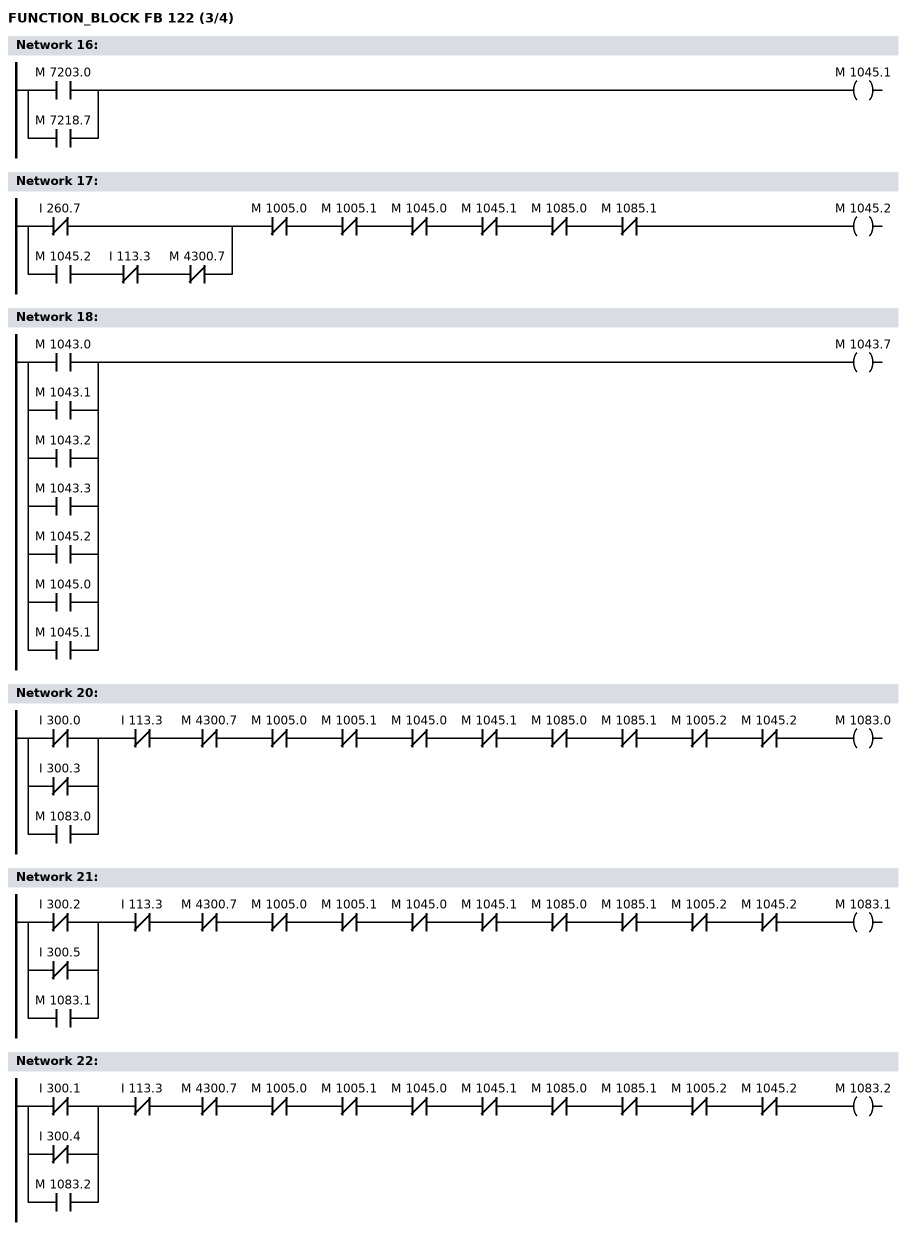

      O     M   7203.0;
      O     M   7218.7;
      =     M   1045.1;
NETWORK
TITLE =

      A(    ;
      ON    I    260.7;
      O     ;
      A     M   1045.2;
      AN    I    113.3;
      AN    M   4300.7;
      )     ;
      AN    M   1005.0;
      AN    M   1005.1;
      AN    M   1045.0;
      AN    M   1045.1;
      AN    M   1085.0;
      AN    M   1085.1;
      =     M   1045.2;
NETWORK
TITLE =

      O     M   1043.0;
      O     M   1043.1;
      O     M   1043.2;
      O     M   1043.3;
      O     M   1045.2;
      O     M   1045.0;
      O     M   1045.1;
      =     M   1043.7;
NETWORK
TITLE =리턴3 이상

NETWORK
TITLE =

      A(    ;
      ON    I    300.0;
      ON    I    300.3;
      O     M   1083.0;
      )     ;
      AN    I    113.3;
      AN    M   4300.7;
      AN    M   1005.0;
      AN    M   1005.1;
      AN    M   1045.0;
      AN    M   1045.1;
      AN    M   1085.0;
      AN    M   1085.1;
      AN    M   1005.2;
      AN    M   1045.2;
      =     M   1083.0;
NETWORK
TITLE =

      A(    ;
      ON    I    300.2;
      ON    I    300.5;
      O     M   1083.1;
      )     ;
      AN    I    113.3;
      AN    M   4300.7;
      AN    M   1005.0;
      AN    M   1005.1;
      AN    M   1045.0;
      AN    M   1045.1;
      AN    M   1085.0;
      AN    M   1085.1;
      AN    M   1005.2;
      AN    M   1045.2;
      =     M   1083.1;
NETWORK
TITLE =

      A(    ;
      ON    I    300.1;
      ON    I    300.4;
      O     M   1083.2;
      )     ;
      AN    I    113.3;
      AN    M   4300.7;
      AN    M   1005.0;
      AN    M   1005.1;
      AN    M   1045.0;
      AN    M   1045.1;
      AN    M   1085.0;
      AN    M   1085.1;
      AN    M   1005.2;
      AN    M   1045.2;
      =     M   1083.2;
NETWORK
TITLE =
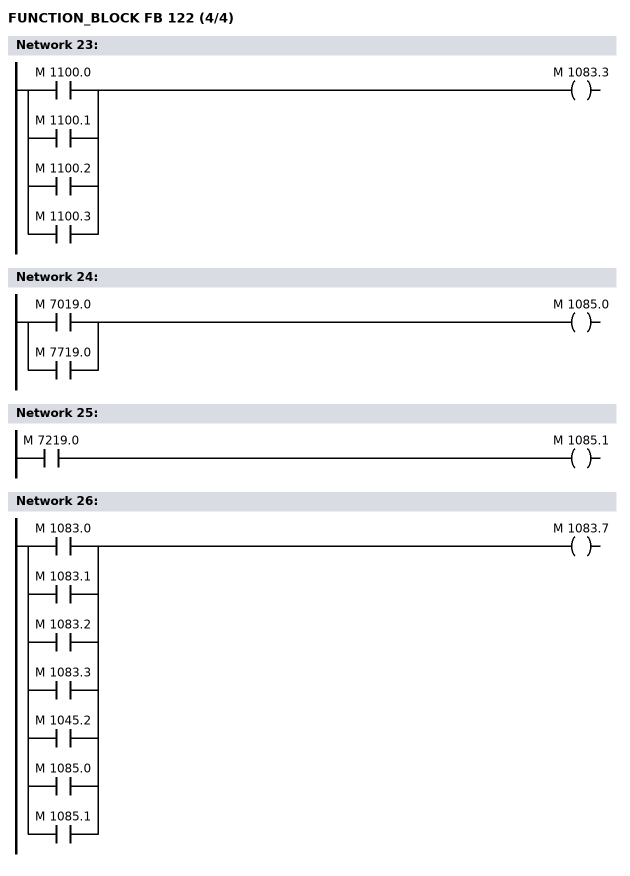

      O     M   1100.0;
      O     M   1100.1;
      O     M   1100.2;
      O     M   1100.3;
      =     M   1083.3;
NETWORK
TITLE =

      O     M   7019.0;
      O     M   7719.0;
      =     M   1085.0;
NETWORK
TITLE =

      A     M   7219.0;
      =     M   1085.1;
NETWORK
TITLE =

      O     M   1083.0;
      O     M   1083.1;
      O     M   1083.2;
      O     M   1083.3;
      O     M   1045.2;
      O     M   1085.0;
      O     M   1085.1;
      =     M   1083.7;
END_FUNCTION_BLOCK

DATA_BLOCK DB 122
TITLE =
VERSION : 0.0

 FB 122
BEGIN
END_DATA_BLOCK

FUNCTION FC 122 : VOID
TITLE =
VERSION : 0.1

BEGIN
NETWORK
TITLE =리턴1 SOL동작관련

NETWORK
TITLE =
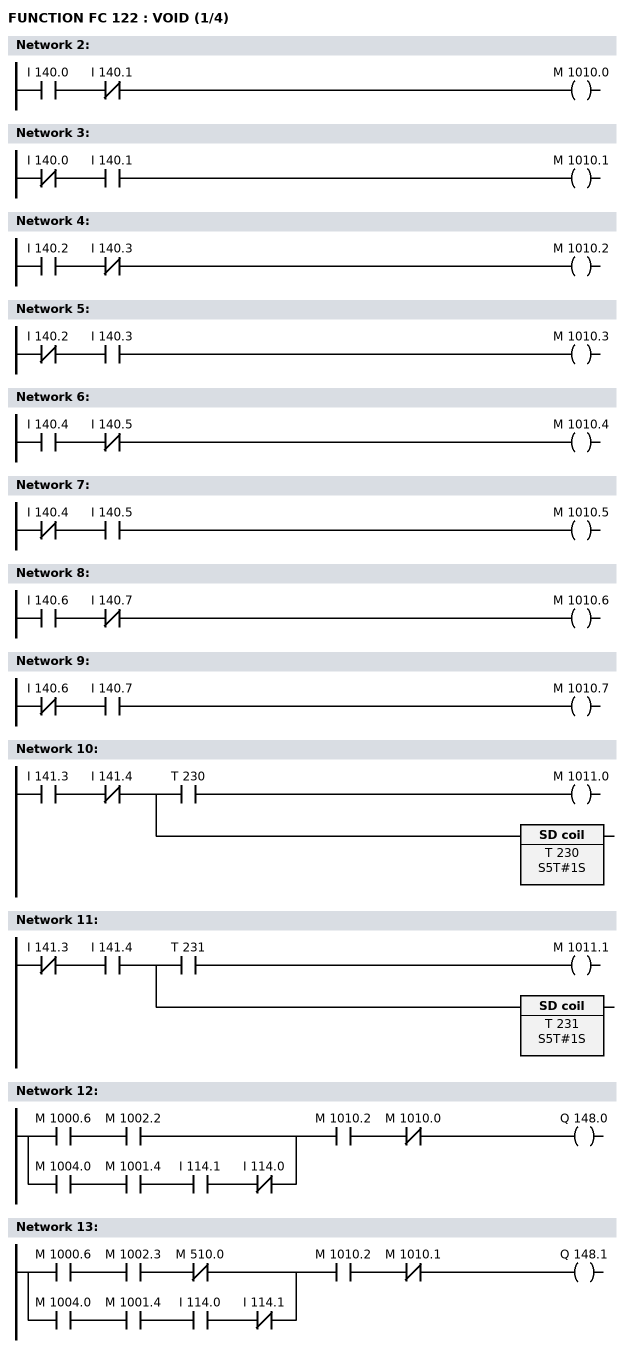

      A     I    140.0;
      AN    I    140.1;
      =     M   1010.0;
NETWORK
TITLE =

      AN    I    140.0;
      A     I    140.1;
      =     M   1010.1;
NETWORK
TITLE =

      A     I    140.2;
      AN    I    140.3;
      =     M   1010.2;
NETWORK
TITLE =

      AN    I    140.2;
      A     I    140.3;
      =     M   1010.3;
NETWORK
TITLE =

      A     I    140.4;
      AN    I    140.5;
      =     M   1010.4;
NETWORK
TITLE =

      AN    I    140.4;
      A     I    140.5;
      =     M   1010.5;
NETWORK
TITLE =

      A     I    140.6;
      AN    I    140.7;
      =     M   1010.6;
NETWORK
TITLE =

      AN    I    140.6;
      A     I    140.7;
      =     M   1010.7;
NETWORK
TITLE =

      A     I    141.3;
      AN    I    141.4;
      =     L      0.0;
      A     L      0.0;
      A     T    230;
      =     M   1011.0;
      A     L      0.0;
      BLD   102;
      L     S5T#1S;
      SD    T    230;
NETWORK
TITLE =

      AN    I    141.3;
      A     I    141.4;
      =     L      0.0;
      A     L      0.0;
      A     T    231;
      =     M   1011.1;
      A     L      0.0;
      BLD   102;
      L     S5T#1S;
      SD    T    231;
NETWORK
TITLE =

      A(    ;
      A     M   1000.6;
      A     M   1002.2;
      O     ;
      A     M   1004.0;
      A     M   1001.4;
      A     I    114.1;
      AN    I    114.0;
      )     ;
      A     M   1010.2;
      AN    M   1010.0;
      =     Q    148.0;
NETWORK
TITLE =

      A(    ;
      A     M   1000.6;
      A     M   1002.3;
      AN    M    510.0;
      O     ;
      A     M   1004.0;
      A     M   1001.4;
      A     I    114.0;
      AN    I    114.1;
      )     ;
      A     M   1010.2;
      AN    M   1010.1;
      =     Q    148.1;
NETWORK
TITLE =
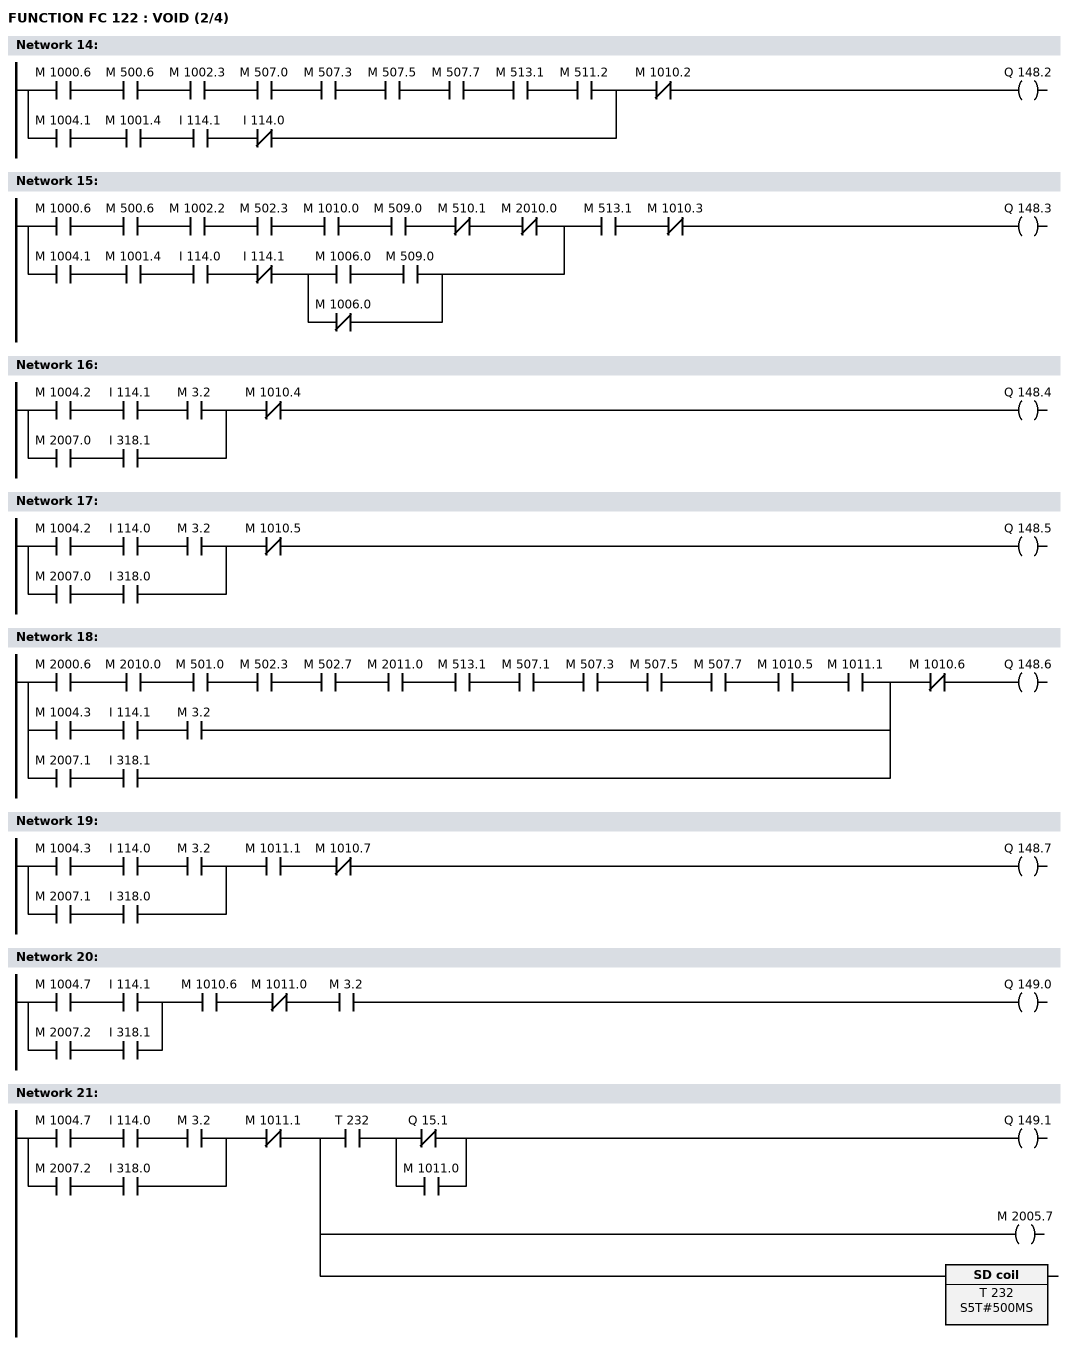

      A(    ;
      A     M   1000.6;
      A     M    500.6;
      A     M   1002.3;
      A     M    507.0;
      A     M    507.3;
      A     M    507.5;
      A     M    507.7;
      A     M    513.1;
      A     M    511.2;
      O     ;
      A     M   1004.1;
      A     M   1001.4;
      A     I    114.1;
      AN    I    114.0;
      )     ;
      AN    M   1010.2;
      =     Q    148.2;
NETWORK
TITLE =

      A(    ;
      A     M   1000.6;
      A     M    500.6;
      A     M   1002.2;
      A     M    502.3;
      A     M   1010.0;
      A     M    509.0;
      AN    M    510.1;
      AN    M   2010.0;
      O     ;
      A     M   1004.1;
      A     M   1001.4;
      A     I    114.0;
      AN    I    114.1;
      A(    ;
      A     M   1006.0;
      A     M    509.0;
      ON    M   1006.0;
      )     ;
      )     ;
      A     M    513.1;
      AN    M   1010.3;
      =     Q    148.3;
NETWORK
TITLE =

      A(    ;
      A     M   1004.2;
      A     I    114.1;
      A     M      3.2;
      O     ;
      A     M   2007.0;
      A     I    318.1;
      )     ;
      AN    M   1010.4;
      =     Q    148.4;
NETWORK
TITLE =

      A(    ;
      A     M   1004.2;
      A     I    114.0;
      A     M      3.2;
      O     ;
      A     M   2007.0;
      A     I    318.0;
      )     ;
      AN    M   1010.5;
      =     Q    148.5;
NETWORK
TITLE =

      A(    ;
      A     M   2000.6;
      A     M   2010.0;
      A     M    501.0;
      A     M    502.3;
      A     M    502.7;
      A     M   2011.0;
      A     M    513.1;
      A     M    507.1;
      A     M    507.3;
      A     M    507.5;
      A     M    507.7;
      A     M   1010.5;
      A     M   1011.1;
      O     ;
      A     M   1004.3;
      A     I    114.1;
      A     M      3.2;
      O     ;
      A     M   2007.1;
      A     I    318.1;
      )     ;
      AN    M   1010.6;
      =     Q    148.6;
NETWORK
TITLE =

      A(    ;
      A     M   1004.3;
      A     I    114.0;
      A     M      3.2;
      O     ;
      A     M   2007.1;
      A     I    318.0;
      )     ;
      A     M   1011.1;
      AN    M   1010.7;
      =     Q    148.7;
NETWORK
TITLE =

      A(    ;
      A     M   1004.7;
      A     I    114.1;
      O     ;
      A     M   2007.2;
      A     I    318.1;
      )     ;
      A     M   1010.6;
      AN    M   1011.0;
      A     M      3.2;
      =     Q    149.0;
NETWORK
TITLE =

      A(    ;
      A     M   1004.7;
      A     I    114.0;
      A     M      3.2;
      O     ;
      A     M   2007.2;
      A     I    318.0;
      )     ;
      AN    M   1011.1;
      =     L      0.0;
      A     L      0.0;
      A     T    232;
      A(    ;
      ON    Q     15.1;
      O     M   1011.0;
      )     ;
      =     Q    149.1;
      A     L      0.0;
      BLD   102;
      =     M   2005.7;
      A     L      0.0;
      BLD   102;
      L     S5T#500MS;
      SD    T    232;
NETWORK
TITLE =
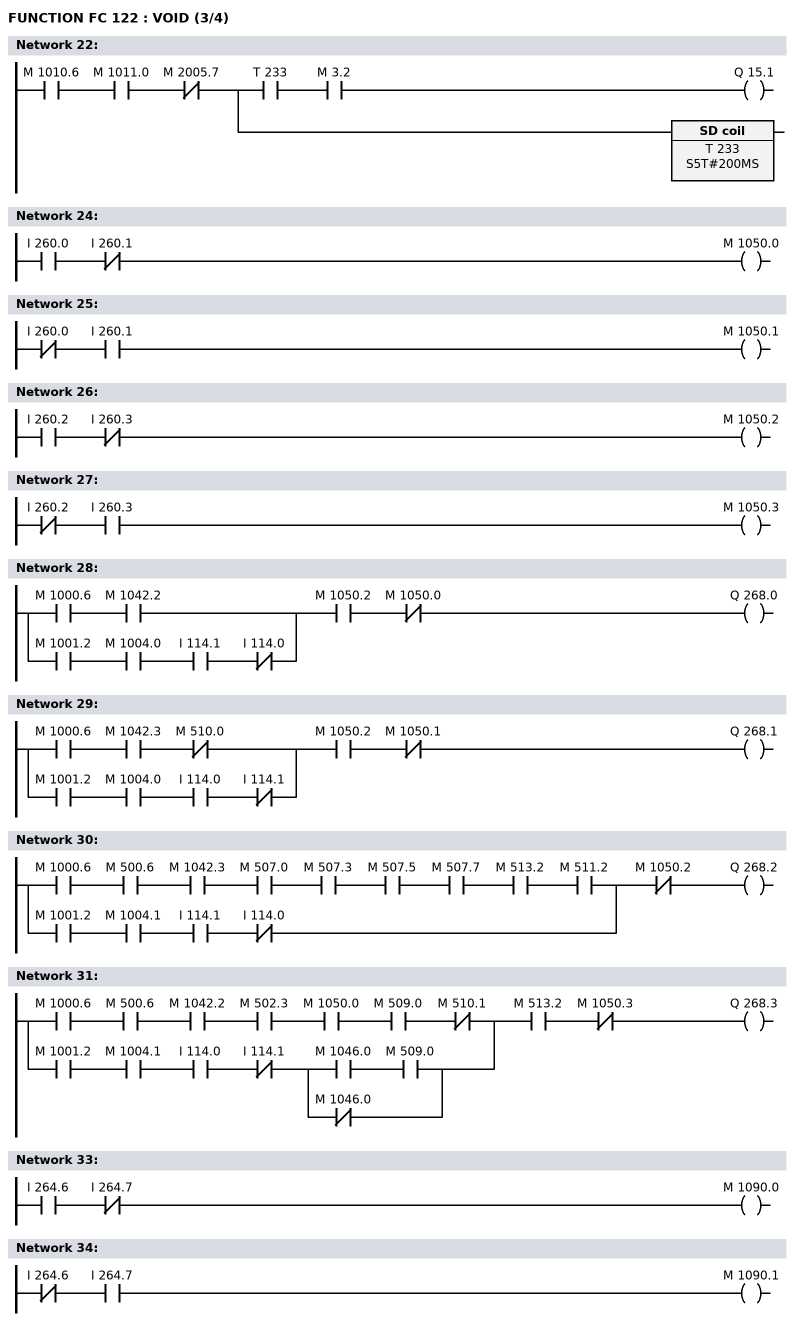

      A     M   1010.6;
      A     M   1011.0;
      AN    M   2005.7;
      =     L      0.0;
      A     L      0.0;
      A     T    233;
      A     M      3.2;
      =     Q     15.1;
      A     L      0.0;
      BLD   102;
      L     S5T#200MS;
      SD    T    233;
NETWORK
TITLE =RETURN2 SOL동작관련

NETWORK
TITLE =

      A     I    260.0;
      AN    I    260.1;
      =     M   1050.0;
NETWORK
TITLE =

      AN    I    260.0;
      A     I    260.1;
      =     M   1050.1;
NETWORK
TITLE =

      A     I    260.2;
      AN    I    260.3;
      =     M   1050.2;
NETWORK
TITLE =

      AN    I    260.2;
      A     I    260.3;
      =     M   1050.3;
NETWORK
TITLE =

      A(    ;
      A     M   1000.6;
      A     M   1042.2;
      O     ;
      A     M   1001.2;
      A     M   1004.0;
      A     I    114.1;
      AN    I    114.0;
      )     ;
      A     M   1050.2;
      AN    M   1050.0;
      =     Q    268.0;
NETWORK
TITLE =

      A(    ;
      A     M   1000.6;
      A     M   1042.3;
      AN    M    510.0;
      O     ;
      A     M   1001.2;
      A     M   1004.0;
      A     I    114.0;
      AN    I    114.1;
      )     ;
      A     M   1050.2;
      AN    M   1050.1;
      =     Q    268.1;
NETWORK
TITLE =

      A(    ;
      A     M   1000.6;
      A     M    500.6;
      A     M   1042.3;
      A     M    507.0;
      A     M    507.3;
      A     M    507.5;
      A     M    507.7;
      A     M    513.2;
      A     M    511.2;
      O     ;
      A     M   1001.2;
      A     M   1004.1;
      A     I    114.1;
      AN    I    114.0;
      )     ;
      AN    M   1050.2;
      =     Q    268.2;
NETWORK
TITLE =

      A(    ;
      A     M   1000.6;
      A     M    500.6;
      A     M   1042.2;
      A     M    502.3;
      A     M   1050.0;
      A     M    509.0;
      AN    M    510.1;
      O     ;
      A     M   1001.2;
      A     M   1004.1;
      A     I    114.0;
      AN    I    114.1;
      A(    ;
      A     M   1046.0;
      A     M    509.0;
      ON    M   1046.0;
      )     ;
      )     ;
      A     M    513.2;
      AN    M   1050.3;
      =     Q    268.3;
NETWORK
TITLE =RETURN3 SOL동작관련

NETWORK
TITLE =

      A     I    264.6;
      AN    I    264.7;
      =     M   1090.0;
NETWORK
TITLE =

      AN    I    264.6;
      A     I    264.7;
      =     M   1090.1;
NETWORK
TITLE =
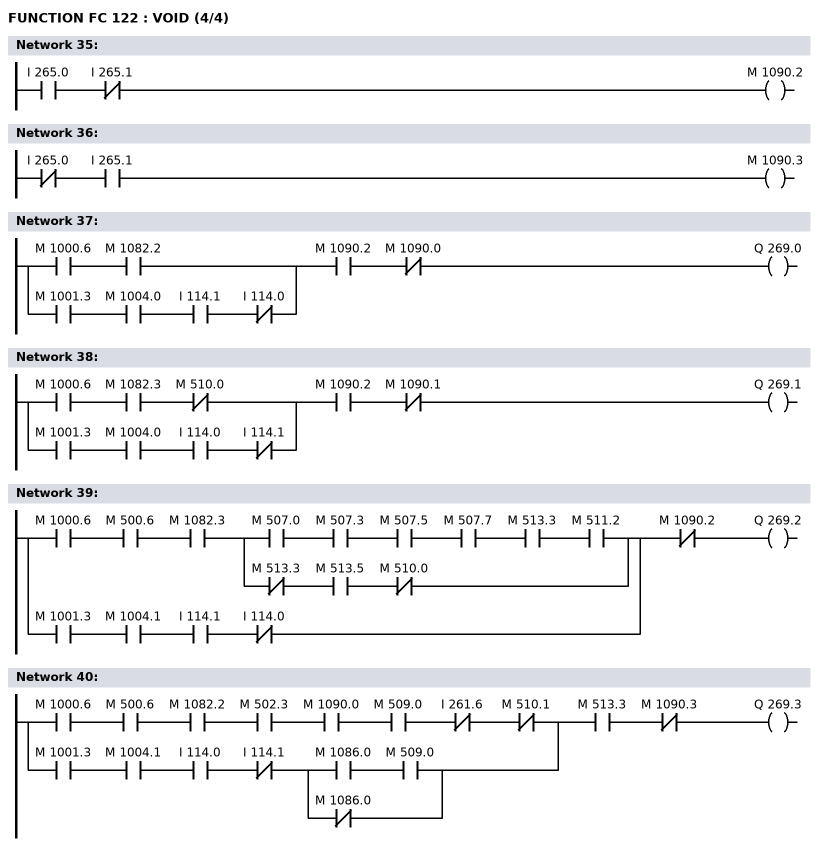

      A     I    265.0;
      AN    I    265.1;
      =     M   1090.2;
NETWORK
TITLE =

      AN    I    265.0;
      A     I    265.1;
      =     M   1090.3;
NETWORK
TITLE =

      A(    ;
      A     M   1000.6;
      A     M   1082.2;
      O     ;
      A     M   1001.3;
      A     M   1004.0;
      A     I    114.1;
      AN    I    114.0;
      )     ;
      A     M   1090.2;
      AN    M   1090.0;
      =     Q    269.0;
NETWORK
TITLE =

      A(    ;
      A     M   1000.6;
      A     M   1082.3;
      AN    M    510.0;
      O     ;
      A     M   1001.3;
      A     M   1004.0;
      A     I    114.0;
      AN    I    114.1;
      )     ;
      A     M   1090.2;
      AN    M   1090.1;
      =     Q    269.1;
NETWORK
TITLE =

      A(    ;
      A     M   1000.6;
      A     M    500.6;
      A     M   1082.3;
      A(    ;
      A     M    507.0;
      A     M    507.3;
      A     M    507.5;
      A     M    507.7;
      A     M    513.3;
      A     M    511.2;
      O     ;
      AN    M    513.3;
      A     M    513.5;
      AN    M    510.0;
      )     ;
      O     ;
      A     M   1001.3;
      A     M   1004.1;
      A     I    114.1;
      AN    I    114.0;
      )     ;
      AN    M   1090.2;
      =     Q    269.2;
NETWORK
TITLE =

      A(    ;
      A     M   1000.6;
      A     M    500.6;
      A     M   1082.2;
      A     M    502.3;
      A     M   1090.0;
      A     M    509.0;
      AN    I    261.6;
      AN    M    510.1;
      O     ;
      A     M   1001.3;
      A     M   1004.1;
      A     I    114.0;
      AN    I    114.1;
      A(    ;
      A     M   1086.0;
      A     M    509.0;
      ON    M   1086.0;
      )     ;
      )     ;
      A     M    513.3;
      AN    M   1090.3;
      =     Q    269.3;
END_FUNCTION

FUNCTION FC 123 : VOID
TITLE =
VERSION : 0.1

BEGIN
NETWORK
TITLE =
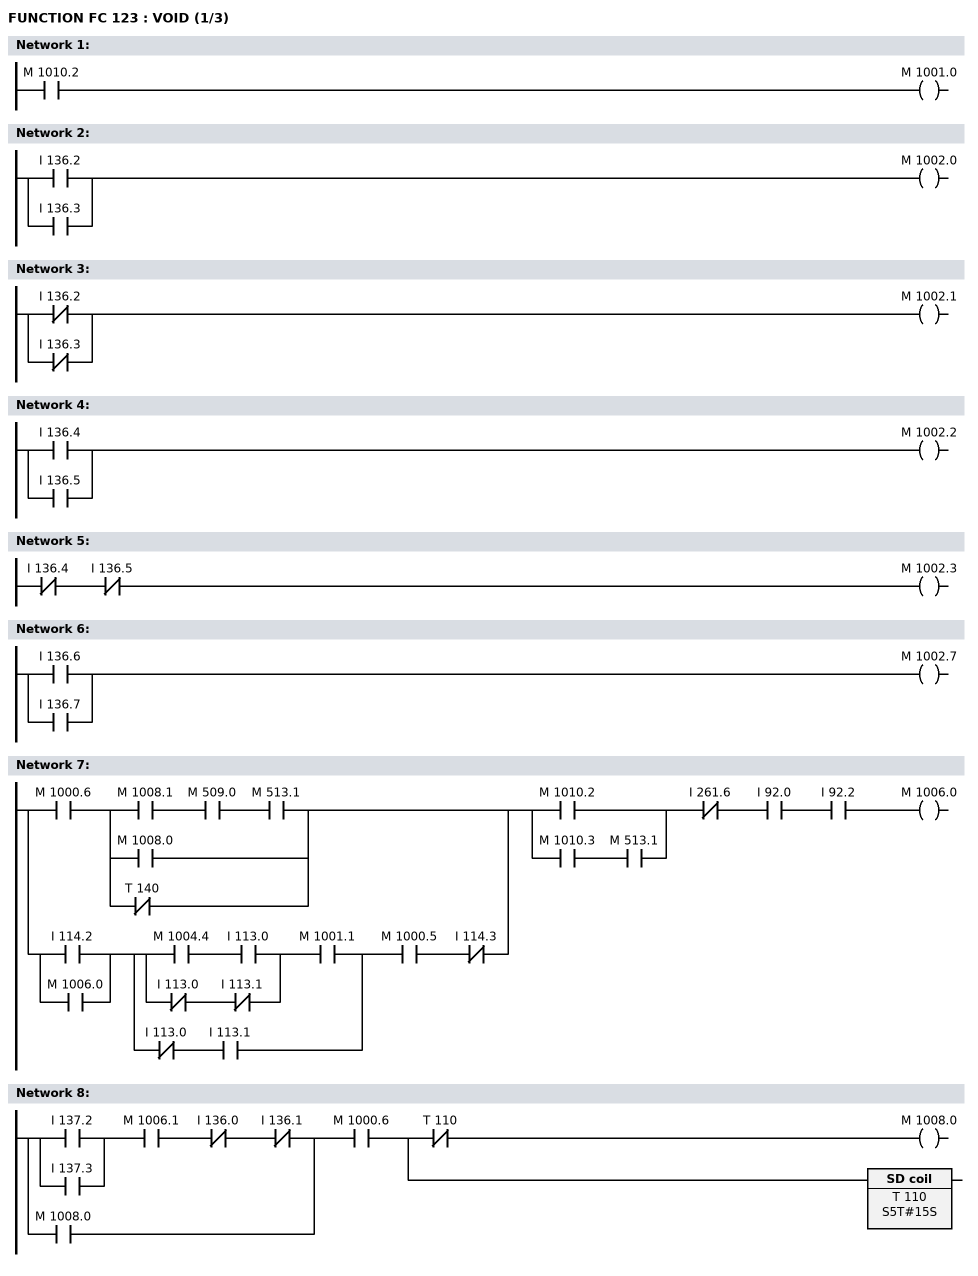

      A     M   1010.2;
      =     M   1001.0;
NETWORK
TITLE =

      O     I    136.2;
      O     I    136.3;
      =     M   1002.0;
NETWORK
TITLE =

      ON    I    136.2;
      ON    I    136.3;
      =     M   1002.1;
NETWORK
TITLE =

      O     I    136.4;
      O     I    136.5;
      =     M   1002.2;
NETWORK
TITLE =

      AN    I    136.4;
      AN    I    136.5;
      =     M   1002.3;
NETWORK
TITLE =

      O     I    136.6;
      O     I    136.7;
      =     M   1002.7;
NETWORK
TITLE =

      A(    ;
      A     M   1000.6;
      A(    ;
      A     M   1008.1;
      A     M    509.0;
      A     M    513.1;
      O     M   1008.0;
      ON    T    140;
      )     ;
      O     ;
      A(    ;
      O     I    114.2;
      O     M   1006.0;
      )     ;
      A(    ;
      A(    ;
      A     M   1004.4;
      A     I    113.0;
      O     ;
      AN    I    113.0;
      AN    I    113.1;
      )     ;
      A     M   1001.1;
      O     ;
      AN    I    113.0;
      A     I    113.1;
      )     ;
      A     M   1000.5;
      AN    I    114.3;
      )     ;
      A(    ;
      O     M   1010.2;
      O     ;
      A     M   1010.3;
      A     M    513.1;
      )     ;
      AN    I    261.6;
      A     I     92.0;
      A     I     92.2;
      =     M   1006.0;
NETWORK
TITLE =

      A(    ;
      A(    ;
      O     I    137.2;
      O     I    137.3;
      )     ;
      A     M   1006.1;
      AN    I    136.0;
      AN    I    136.1;
      O     M   1008.0;
      )     ;
      A     M   1000.6;
      =     L      0.0;
      A     L      0.0;
      AN    T    110;
      =     M   1008.0;
      A     L      0.0;
      BLD   102;
      L     S5T#15S;
      SD    T    110;
NETWORK
TITLE =
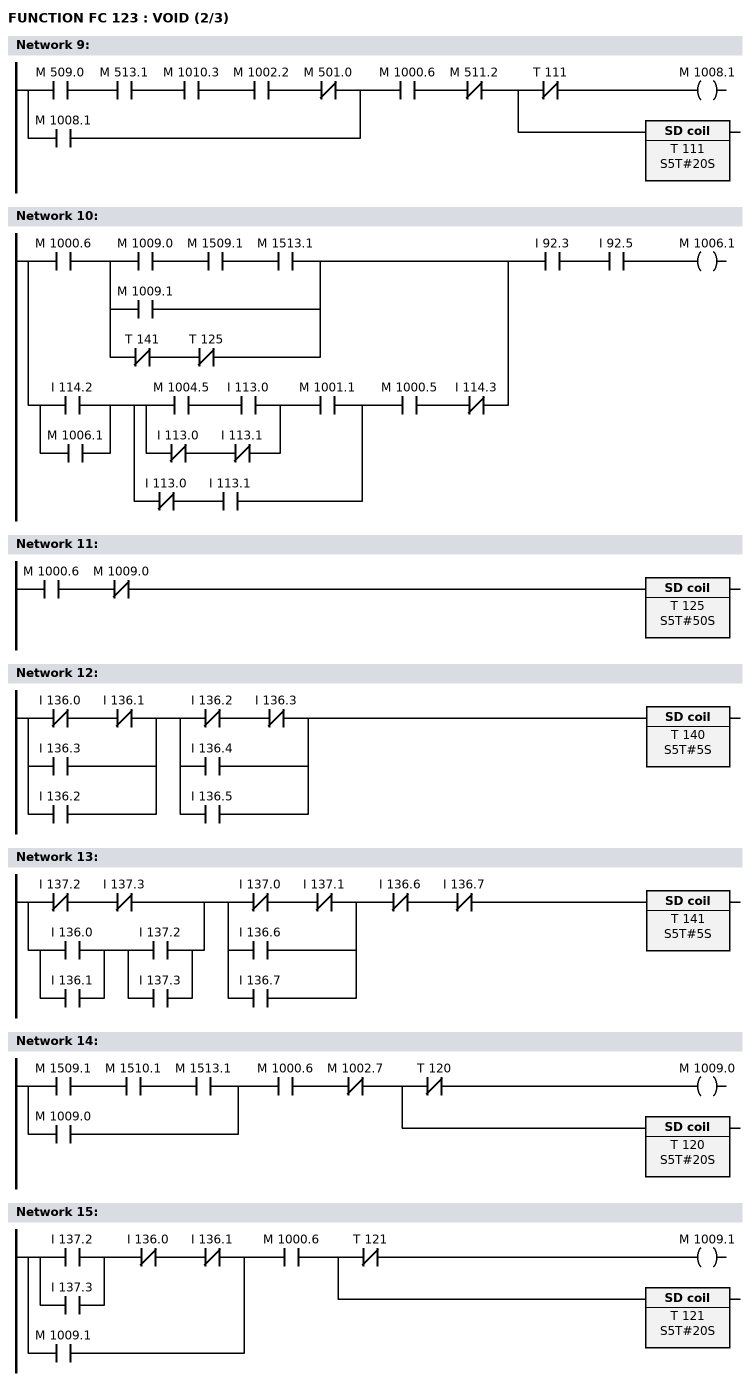

      A(    ;
      A     M    509.0;
      A     M    513.1;
      A     M   1010.3;
      A     M   1002.2;
      AN    M    501.0;
      O     M   1008.1;
      )     ;
      A     M   1000.6;
      AN    M    511.2;
      =     L      0.0;
      A     L      0.0;
      AN    T    111;
      =     M   1008.1;
      A     L      0.0;
      BLD   102;
      L     S5T#20S;
      SD    T    111;
NETWORK
TITLE =

      A(    ;
      A     M   1000.6;
      A(    ;
      A     M   1009.0;
      A     M   1509.1;
      A     M   1513.1;
      O     M   1009.1;
      O     ;
      AN    T    141;
      AN    T    125;
      )     ;
      O     ;
      A(    ;
      O     I    114.2;
      O     M   1006.1;
      )     ;
      A(    ;
      A(    ;
      A     M   1004.5;
      A     I    113.0;
      O     ;
      AN    I    113.0;
      AN    I    113.1;
      )     ;
      A     M   1001.1;
      O     ;
      AN    I    113.0;
      A     I    113.1;
      )     ;
      A     M   1000.5;
      AN    I    114.3;
      )     ;
      A     I     92.3;
      A     I     92.5;
      =     M   1006.1;
NETWORK
TITLE =

      A     M   1000.6;
      AN    M   1009.0;
      L     S5T#50S;
      SD    T    125;
NETWORK
TITLE =

      A(    ;
      AN    I    136.0;
      AN    I    136.1;
      O     I    136.3;
      O     I    136.2;
      )     ;
      A(    ;
      AN    I    136.2;
      AN    I    136.3;
      O     I    136.4;
      O     I    136.5;
      )     ;
      L     S5T#5S;
      SD    T    140;
NETWORK
TITLE =

      A(    ;
      AN    I    137.2;
      AN    I    137.3;
      O     ;
      A(    ;
      O     I    136.0;
      O     I    136.1;
      )     ;
      A(    ;
      O     I    137.2;
      O     I    137.3;
      )     ;
      )     ;
      A(    ;
      AN    I    137.0;
      AN    I    137.1;
      O     I    136.6;
      O     I    136.7;
      )     ;
      AN    I    136.6;
      AN    I    136.7;
      L     S5T#5S;
      SD    T    141;
NETWORK
TITLE =

      A(    ;
      A     M   1509.1;
      A     M   1510.1;
      A     M   1513.1;
      O     M   1009.0;
      )     ;
      A     M   1000.6;
      AN    M   1002.7;
      =     L      0.0;
      A     L      0.0;
      AN    T    120;
      =     M   1009.0;
      A     L      0.0;
      BLD   102;
      L     S5T#20S;
      SD    T    120;
NETWORK
TITLE =

      A(    ;
      A(    ;
      O     I    137.2;
      O     I    137.3;
      )     ;
      AN    I    136.0;
      AN    I    136.1;
      O     M   1009.1;
      )     ;
      A     M   1000.6;
      =     L      0.0;
      A     L      0.0;
      AN    T    121;
      =     M   1009.1;
      A     L      0.0;
      BLD   102;
      L     S5T#20S;
      SD    T    121;
NETWORK
TITLE =
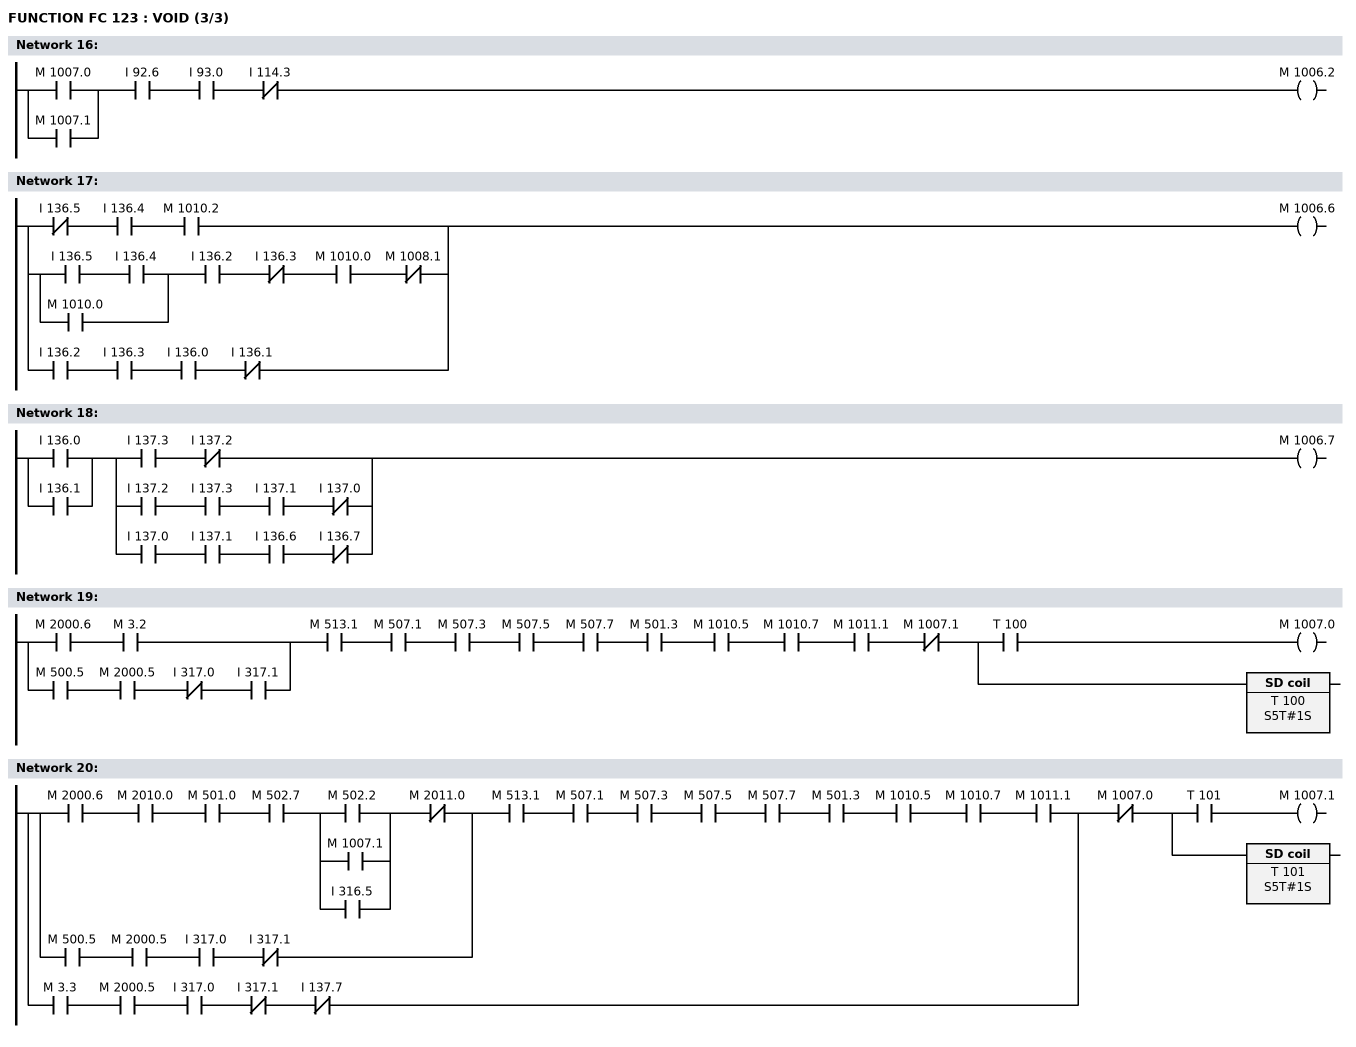

      A(    ;
      O     M   1007.0;
      O     M   1007.1;
      )     ;
      A     I     92.6;
      A     I     93.0;
      AN    I    114.3;
      =     M   1006.2;
NETWORK
TITLE =

      AN    I    136.5;
      A     I    136.4;
      A     M   1010.2;
      O     ;
      A(    ;
      A     I    136.5;
      A     I    136.4;
      O     M   1010.0;
      )     ;
      A     I    136.2;
      AN    I    136.3;
      A     M   1010.0;
      AN    M   1008.1;
      O     ;
      A     I    136.2;
      A     I    136.3;
      A     I    136.0;
      AN    I    136.1;
      =     M   1006.6;
NETWORK
TITLE =

      A(    ;
      O     I    136.0;
      O     I    136.1;
      )     ;
      A(    ;
      A     I    137.3;
      AN    I    137.2;
      O     ;
      A     I    137.2;
      A     I    137.3;
      A     I    137.1;
      AN    I    137.0;
      O     ;
      A     I    137.0;
      A     I    137.1;
      A     I    136.6;
      AN    I    136.7;
      )     ;
      =     M   1006.7;
NETWORK
TITLE =

      A(    ;
      A     M   2000.6;
      A     M      3.2;
      O     ;
      A     M    500.5;
      A     M   2000.5;
      AN    I    317.0;
      A     I    317.1;
      )     ;
      A     M    513.1;
      A     M    507.1;
      A     M    507.3;
      A     M    507.5;
      A     M    507.7;
      A     M    501.3;
      A     M   1010.5;
      A     M   1010.7;
      A     M   1011.1;
      AN    M   1007.1;
      =     L      0.0;
      A     L      0.0;
      A     T    100;
      =     M   1007.0;
      A     L      0.0;
      BLD   102;
      L     S5T#1S;
      SD    T    100;
NETWORK
TITLE =

      A(    ;
      A(    ;
      A     M   2000.6;
      A     M   2010.0;
      A     M    501.0;
      A     M    502.7;
      A(    ;
      O     M    502.2;
      O     M   1007.1;
      O     I    316.5;
      )     ;
      AN    M   2011.0;
      O     ;
      A     M    500.5;
      A     M   2000.5;
      A     I    317.0;
      AN    I    317.1;
      )     ;
      A     M    513.1;
      A     M    507.1;
      A     M    507.3;
      A     M    507.5;
      A     M    507.7;
      A     M    501.3;
      A     M   1010.5;
      A     M   1010.7;
      A     M   1011.1;
      O     ;
      A     M      3.3;
      A     M   2000.5;
      A     I    317.0;
      AN    I    317.1;
      AN    I    137.7;
      )     ;
      AN    M   1007.0;
      =     L      0.0;
      A     L      0.0;
      A     T    101;
      =     M   1007.1;
      A     L      0.0;
      BLD   102;
      L     S5T#1S;
      SD    T    101;
END_FUNCTION

FUNCTION FC 124 : VOID
TITLE =
VERSION : 0.1

BEGIN
NETWORK
TITLE =
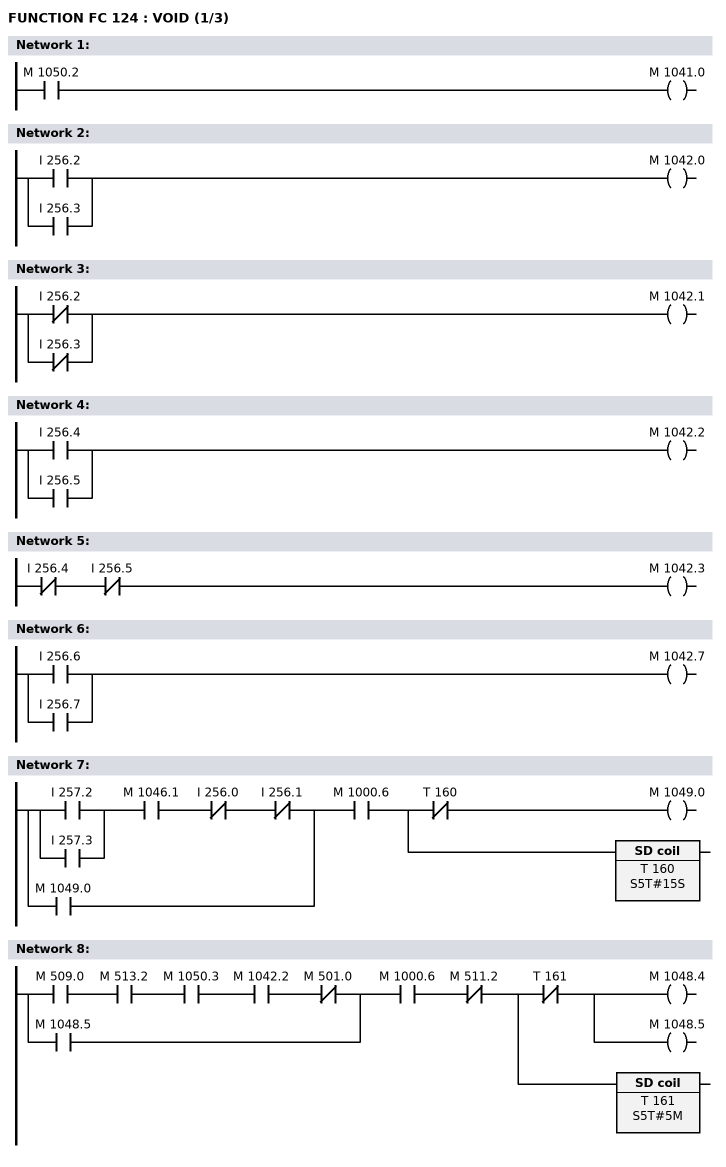

      A     M   1050.2;
      =     M   1041.0;
NETWORK
TITLE =

      O     I    256.2;
      O     I    256.3;
      =     M   1042.0;
NETWORK
TITLE =

      ON    I    256.2;
      ON    I    256.3;
      =     M   1042.1;
NETWORK
TITLE =

      O     I    256.4;
      O     I    256.5;
      =     M   1042.2;
NETWORK
TITLE =

      AN    I    256.4;
      AN    I    256.5;
      =     M   1042.3;
NETWORK
TITLE =

      O     I    256.6;
      O     I    256.7;
      =     M   1042.7;
NETWORK
TITLE =

      A(    ;
      A(    ;
      O     I    257.2;
      O     I    257.3;
      )     ;
      A     M   1046.1;
      AN    I    256.0;
      AN    I    256.1;
      O     M   1049.0;
      )     ;
      A     M   1000.6;
      =     L      0.0;
      A     L      0.0;
      AN    T    160;
      =     M   1049.0;
      A     L      0.0;
      BLD   102;
      L     S5T#15S;
      SD    T    160;
NETWORK
TITLE =

      A(    ;
      A     M    509.0;
      A     M    513.2;
      A     M   1050.3;
      A     M   1042.2;
      AN    M    501.0;
      O     M   1048.5;
      )     ;
      A     M   1000.6;
      AN    M    511.2;
      =     L      0.0;
      A     L      0.0;
      AN    T    161;
      =     M   1048.4;
      =     M   1048.5;
      A     L      0.0;
      BLD   102;
      L     S5T#5M;
      SD    T    161;
NETWORK
TITLE =
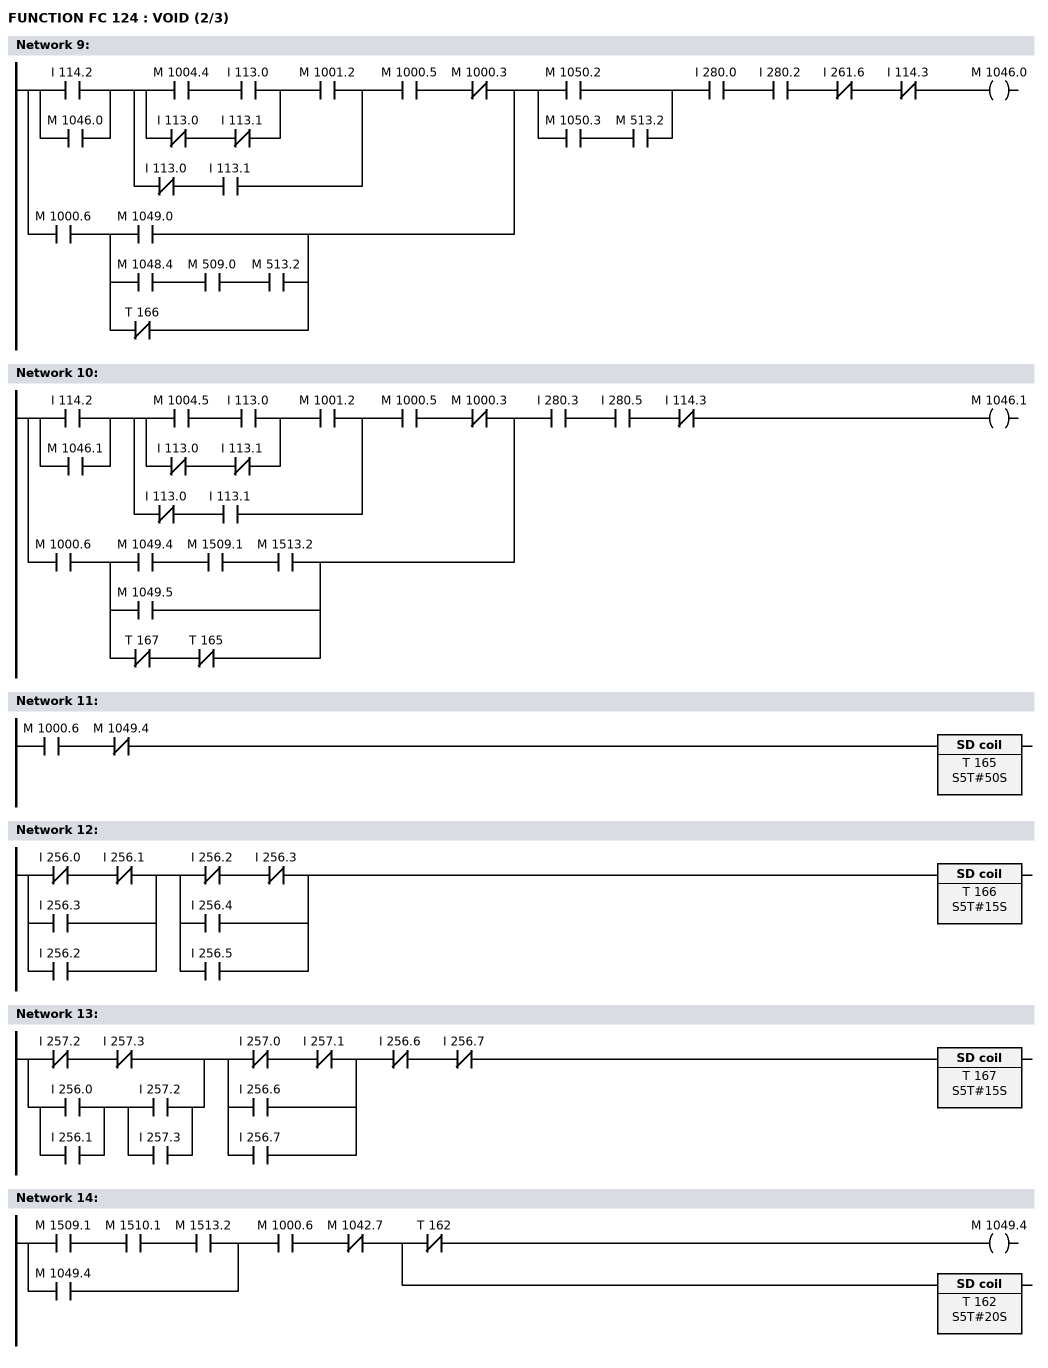

      A(    ;
      A(    ;
      O     I    114.2;
      O     M   1046.0;
      )     ;
      A(    ;
      A(    ;
      A     M   1004.4;
      A     I    113.0;
      O     ;
      AN    I    113.0;
      AN    I    113.1;
      )     ;
      A     M   1001.2;
      O     ;
      AN    I    113.0;
      A     I    113.1;
      )     ;
      A     M   1000.5;
      AN    M   1000.3;
      O     ;
      A     M   1000.6;
      A(    ;
      O     M   1049.0;
      O     ;
      A     M   1048.4;
      A     M    509.0;
      A     M    513.2;
      ON    T    166;
      )     ;
      )     ;
      A(    ;
      O     M   1050.2;
      O     ;
      A     M   1050.3;
      A     M    513.2;
      )     ;
      A     I    280.0;
      A     I    280.2;
      AN    I    261.6;
      AN    I    114.3;
      =     M   1046.0;
NETWORK
TITLE =

      A(    ;
      A(    ;
      O     I    114.2;
      O     M   1046.1;
      )     ;
      A(    ;
      A(    ;
      A     M   1004.5;
      A     I    113.0;
      O     ;
      AN    I    113.0;
      AN    I    113.1;
      )     ;
      A     M   1001.2;
      O     ;
      AN    I    113.0;
      A     I    113.1;
      )     ;
      A     M   1000.5;
      AN    M   1000.3;
      O     ;
      A     M   1000.6;
      A(    ;
      A     M   1049.4;
      A     M   1509.1;
      A     M   1513.2;
      O     M   1049.5;
      O     ;
      AN    T    167;
      AN    T    165;
      )     ;
      )     ;
      A     I    280.3;
      A     I    280.5;
      AN    I    114.3;
      =     M   1046.1;
NETWORK
TITLE =

      A     M   1000.6;
      AN    M   1049.4;
      L     S5T#50S;
      SD    T    165;
NETWORK
TITLE =

      A(    ;
      AN    I    256.0;
      AN    I    256.1;
      O     I    256.3;
      O     I    256.2;
      )     ;
      A(    ;
      AN    I    256.2;
      AN    I    256.3;
      O     I    256.4;
      O     I    256.5;
      )     ;
      L     S5T#15S;
      SD    T    166;
NETWORK
TITLE =

      A(    ;
      AN    I    257.2;
      AN    I    257.3;
      O     ;
      A(    ;
      O     I    256.0;
      O     I    256.1;
      )     ;
      A(    ;
      O     I    257.2;
      O     I    257.3;
      )     ;
      )     ;
      A(    ;
      AN    I    257.0;
      AN    I    257.1;
      O     I    256.6;
      O     I    256.7;
      )     ;
      AN    I    256.6;
      AN    I    256.7;
      L     S5T#15S;
      SD    T    167;
NETWORK
TITLE =

      A(    ;
      A     M   1509.1;
      A     M   1510.1;
      A     M   1513.2;
      O     M   1049.4;
      )     ;
      A     M   1000.6;
      AN    M   1042.7;
      =     L      0.0;
      A     L      0.0;
      AN    T    162;
      =     M   1049.4;
      A     L      0.0;
      BLD   102;
      L     S5T#20S;
      SD    T    162;
NETWORK
TITLE =
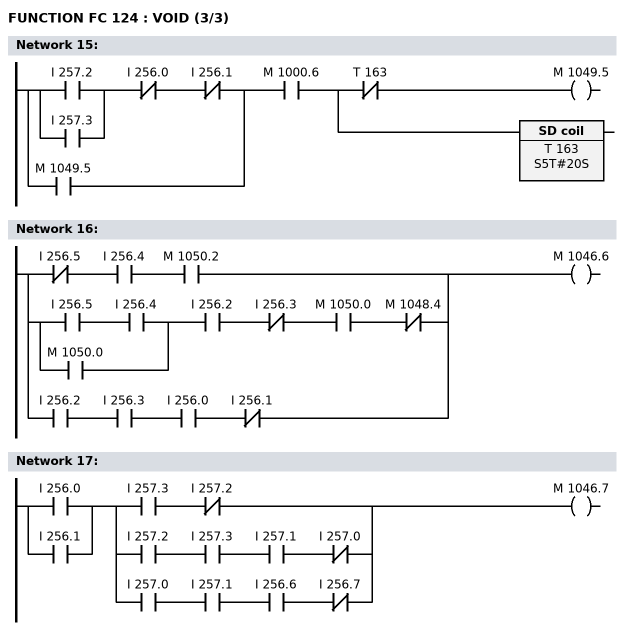

      A(    ;
      A(    ;
      O     I    257.2;
      O     I    257.3;
      )     ;
      AN    I    256.0;
      AN    I    256.1;
      O     M   1049.5;
      )     ;
      A     M   1000.6;
      =     L      0.0;
      A     L      0.0;
      AN    T    163;
      =     M   1049.5;
      A     L      0.0;
      BLD   102;
      L     S5T#20S;
      SD    T    163;
NETWORK
TITLE =

      AN    I    256.5;
      A     I    256.4;
      A     M   1050.2;
      O     ;
      A(    ;
      A     I    256.5;
      A     I    256.4;
      O     M   1050.0;
      )     ;
      A     I    256.2;
      AN    I    256.3;
      A     M   1050.0;
      AN    M   1048.4;
      O     ;
      A     I    256.2;
      A     I    256.3;
      A     I    256.0;
      AN    I    256.1;
      =     M   1046.6;
NETWORK
TITLE =

      A(    ;
      O     I    256.0;
      O     I    256.1;
      )     ;
      A(    ;
      A     I    257.3;
      AN    I    257.2;
      O     ;
      A     I    257.2;
      A     I    257.3;
      A     I    257.1;
      AN    I    257.0;
      O     ;
      A     I    257.0;
      A     I    257.1;
      A     I    256.6;
      AN    I    256.7;
      )     ;
      =     M   1046.7;
END_FUNCTION

FUNCTION FC 125 : VOID
TITLE =
VERSION : 0.1

BEGIN
NETWORK
TITLE =
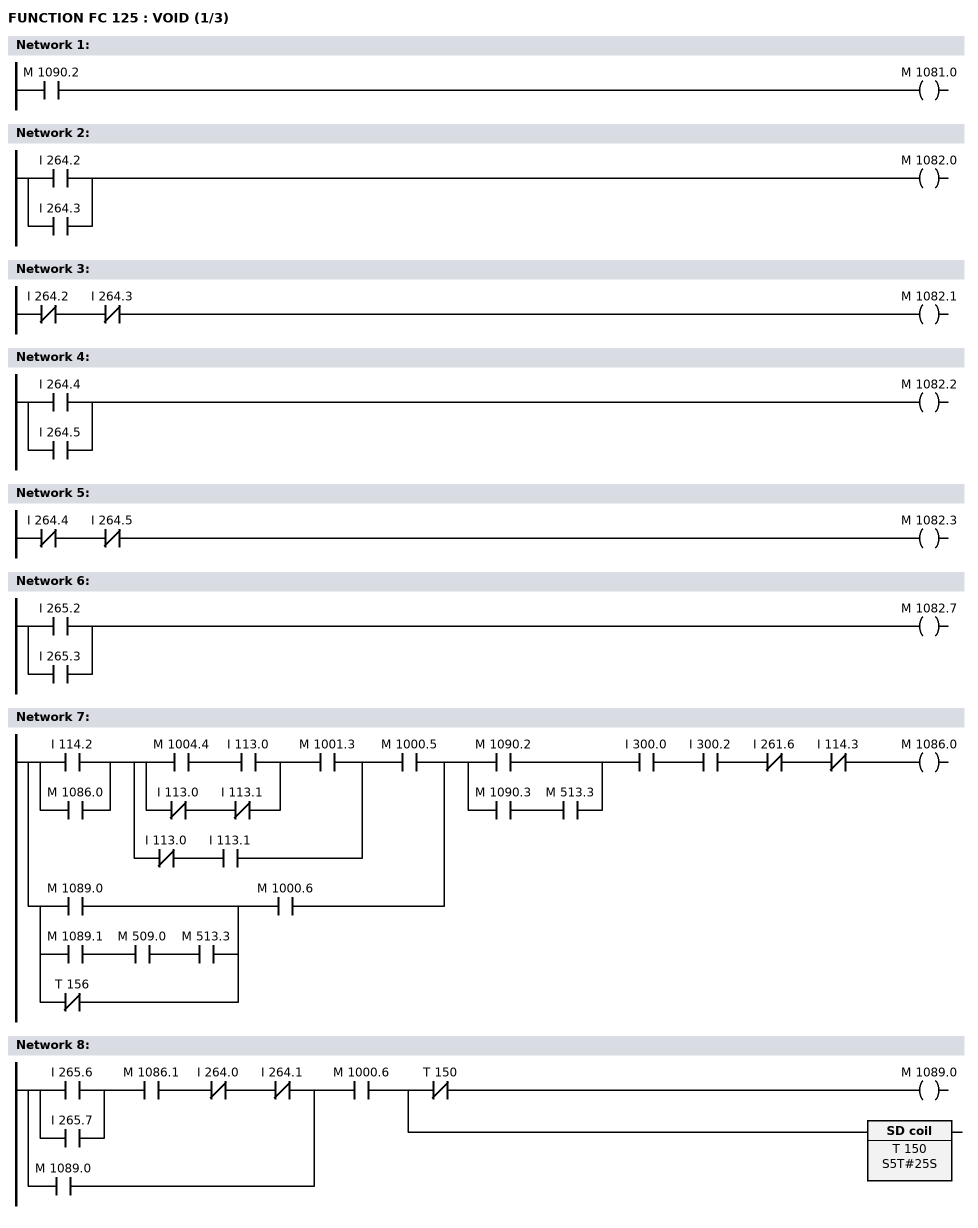

      A     M   1090.2;
      =     M   1081.0;
NETWORK
TITLE =

      O     I    264.2;
      O     I    264.3;
      =     M   1082.0;
NETWORK
TITLE =

      AN    I    264.2;
      AN    I    264.3;
      =     M   1082.1;
NETWORK
TITLE =

      O     I    264.4;
      O     I    264.5;
      =     M   1082.2;
NETWORK
TITLE =

      AN    I    264.4;
      AN    I    264.5;
      =     M   1082.3;
NETWORK
TITLE =

      O     I    265.2;
      O     I    265.3;
      =     M   1082.7;
NETWORK
TITLE =

      A(    ;
      A(    ;
      O     I    114.2;
      O     M   1086.0;
      )     ;
      A(    ;
      A(    ;
      A     M   1004.4;
      A     I    113.0;
      O     ;
      AN    I    113.0;
      AN    I    113.1;
      )     ;
      A     M   1001.3;
      O     ;
      AN    I    113.0;
      A     I    113.1;
      )     ;
      A     M   1000.5;
      O     ;
      A(    ;
      O     M   1089.0;
      O     ;
      A     M   1089.1;
      A     M    509.0;
      A     M    513.3;
      ON    T    156;
      )     ;
      A     M   1000.6;
      )     ;
      A(    ;
      O     M   1090.2;
      O     ;
      A     M   1090.3;
      A     M    513.3;
      )     ;
      A     I    300.0;
      A     I    300.2;
      AN    I    261.6;
      AN    I    114.3;
      =     M   1086.0;
NETWORK
TITLE =

      A(    ;
      A(    ;
      O     I    265.6;
      O     I    265.7;
      )     ;
      A     M   1086.1;
      AN    I    264.0;
      AN    I    264.1;
      O     M   1089.0;
      )     ;
      A     M   1000.6;
      =     L      0.0;
      A     L      0.0;
      AN    T    150;
      =     M   1089.0;
      A     L      0.0;
      BLD   102;
      L     S5T#25S;
      SD    T    150;
NETWORK
TITLE =
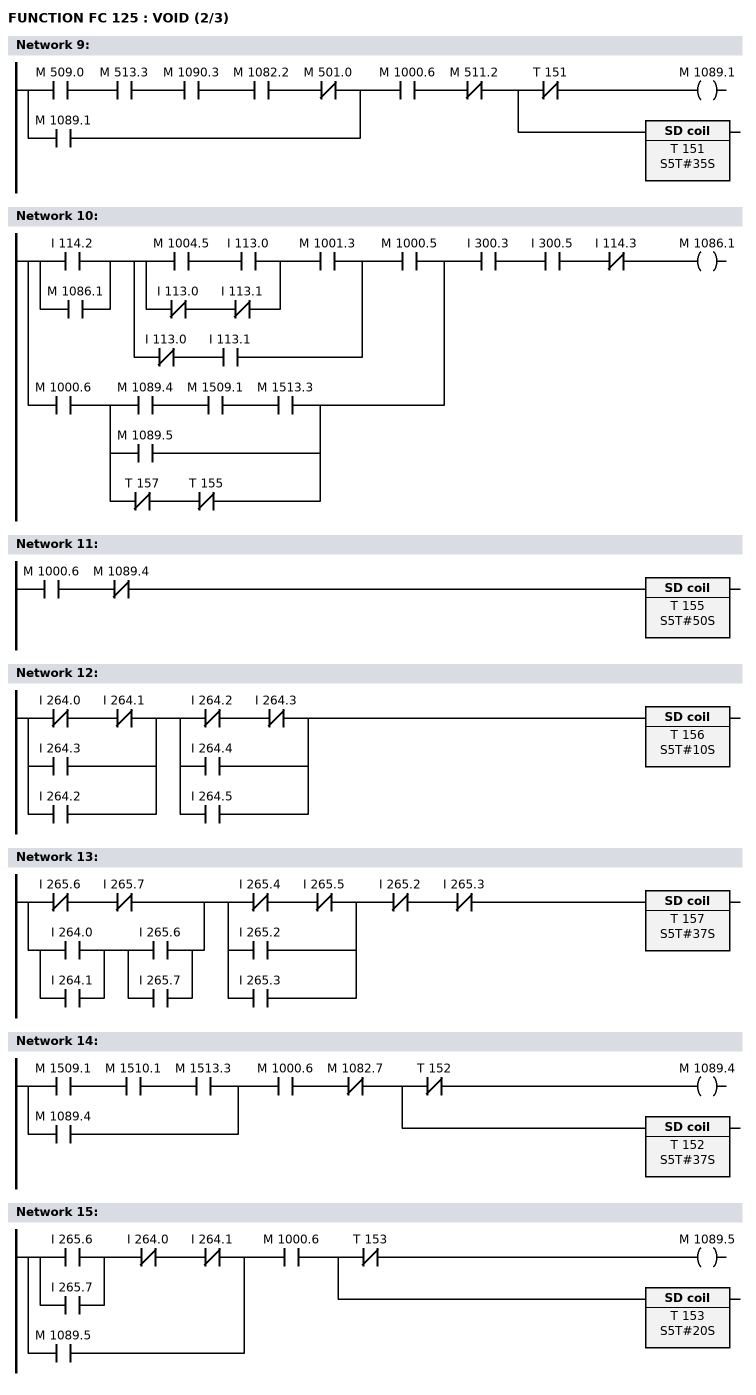

      A(    ;
      A     M    509.0;
      A     M    513.3;
      A     M   1090.3;
      A     M   1082.2;
      AN    M    501.0;
      O     M   1089.1;
      )     ;
      A     M   1000.6;
      AN    M    511.2;
      =     L      0.0;
      A     L      0.0;
      AN    T    151;
      =     M   1089.1;
      A     L      0.0;
      BLD   102;
      L     S5T#35S;
      SD    T    151;
NETWORK
TITLE =

      A(    ;
      A(    ;
      O     I    114.2;
      O     M   1086.1;
      )     ;
      A(    ;
      A(    ;
      A     M   1004.5;
      A     I    113.0;
      O     ;
      AN    I    113.0;
      AN    I    113.1;
      )     ;
      A     M   1001.3;
      O     ;
      AN    I    113.0;
      A     I    113.1;
      )     ;
      A     M   1000.5;
      O     ;
      A     M   1000.6;
      A(    ;
      A     M   1089.4;
      A     M   1509.1;
      A     M   1513.3;
      O     M   1089.5;
      O     ;
      AN    T    157;
      AN    T    155;
      )     ;
      )     ;
      A     I    300.3;
      A     I    300.5;
      AN    I    114.3;
      =     M   1086.1;
NETWORK
TITLE =

      A     M   1000.6;
      AN    M   1089.4;
      L     S5T#50S;
      SD    T    155;
NETWORK
TITLE =

      A(    ;
      AN    I    264.0;
      AN    I    264.1;
      O     I    264.3;
      O     I    264.2;
      )     ;
      A(    ;
      AN    I    264.2;
      AN    I    264.3;
      O     I    264.4;
      O     I    264.5;
      )     ;
      L     S5T#10S;
      SD    T    156;
NETWORK
TITLE =

      A(    ;
      AN    I    265.6;
      AN    I    265.7;
      O     ;
      A(    ;
      O     I    264.0;
      O     I    264.1;
      )     ;
      A(    ;
      O     I    265.6;
      O     I    265.7;
      )     ;
      )     ;
      A(    ;
      AN    I    265.4;
      AN    I    265.5;
      O     I    265.2;
      O     I    265.3;
      )     ;
      AN    I    265.2;
      AN    I    265.3;
      L     S5T#37S;
      SD    T    157;
NETWORK
TITLE =

      A(    ;
      A     M   1509.1;
      A     M   1510.1;
      A     M   1513.3;
      O     M   1089.4;
      )     ;
      A     M   1000.6;
      AN    M   1082.7;
      =     L      0.0;
      A     L      0.0;
      AN    T    152;
      =     M   1089.4;
      A     L      0.0;
      BLD   102;
      L     S5T#37S;
      SD    T    152;
NETWORK
TITLE =

      A(    ;
      A(    ;
      O     I    265.6;
      O     I    265.7;
      )     ;
      AN    I    264.0;
      AN    I    264.1;
      O     M   1089.5;
      )     ;
      A     M   1000.6;
      =     L      0.0;
      A     L      0.0;
      AN    T    153;
      =     M   1089.5;
      A     L      0.0;
      BLD   102;
      L     S5T#20S;
      SD    T    153;
NETWORK
TITLE =
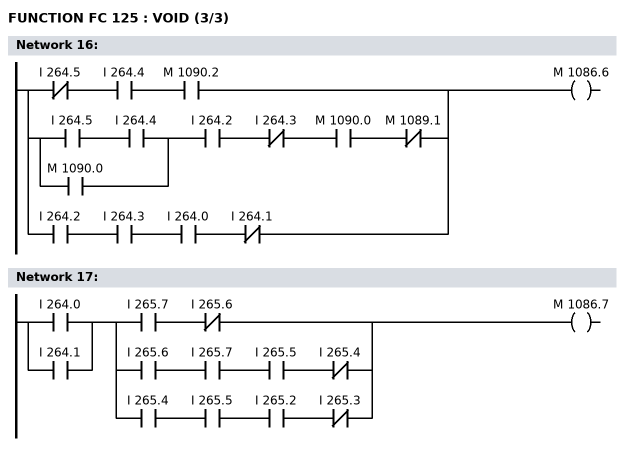

      AN    I    264.5;
      A     I    264.4;
      A     M   1090.2;
      O     ;
      A(    ;
      A     I    264.5;
      A     I    264.4;
      O     M   1090.0;
      )     ;
      A     I    264.2;
      AN    I    264.3;
      A     M   1090.0;
      AN    M   1089.1;
      O     ;
      A     I    264.2;
      A     I    264.3;
      A     I    264.0;
      AN    I    264.1;
      =     M   1086.6;
NETWORK
TITLE =

      A(    ;
      O     I    264.0;
      O     I    264.1;
      )     ;
      A(    ;
      A     I    265.7;
      AN    I    265.6;
      O     ;
      A     I    265.6;
      A     I    265.7;
      A     I    265.5;
      AN    I    265.4;
      O     ;
      A     I    265.4;
      A     I    265.5;
      A     I    265.2;
      AN    I    265.3;
      )     ;
      =     M   1086.7;
END_FUNCTION

FUNCTION FC 126 : VOID
TITLE =
VERSION : 0.1

BEGIN
NETWORK
TITLE =리턴1 인버터 인터록

NETWORK
TITLE =
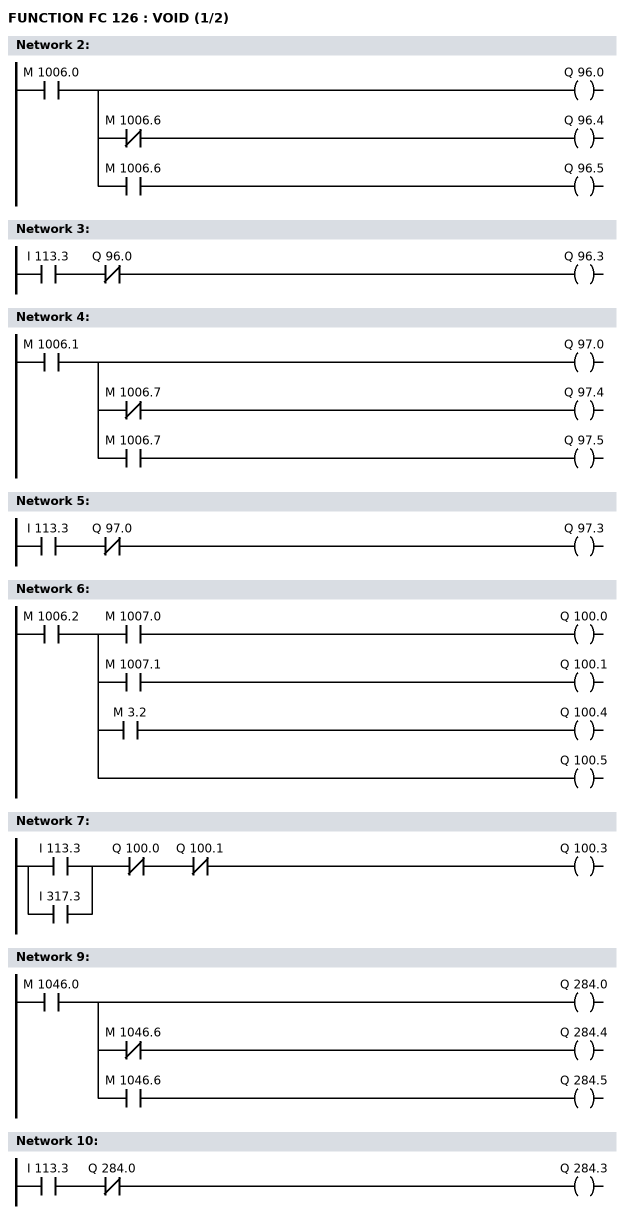

      A     M   1006.0;
      =     L      0.0;
      A     L      0.0;
      BLD   102;
      =     Q     96.0;
      A     L      0.0;
      AN    M   1006.6;
      =     Q     96.4;
      A     L      0.0;
      A     M   1006.6;
      =     Q     96.5;
NETWORK
TITLE =

      A     I    113.3;
      AN    Q     96.0;
      =     Q     96.3;
NETWORK
TITLE =

      A     M   1006.1;
      =     L      0.0;
      A     L      0.0;
      BLD   102;
      =     Q     97.0;
      A     L      0.0;
      AN    M   1006.7;
      =     Q     97.4;
      A     L      0.0;
      A     M   1006.7;
      =     Q     97.5;
NETWORK
TITLE =

      A     I    113.3;
      AN    Q     97.0;
      =     Q     97.3;
NETWORK
TITLE =

      A     M   1006.2;
      =     L      0.0;
      A     L      0.0;
      A     M   1007.0;
      =     Q    100.0;
      A     L      0.0;
      A     M   1007.1;
      =     Q    100.1;
      A     L      0.0;
      A     M      3.2;
      =     Q    100.4;
      A     L      0.0;
      BLD   102;
      =     Q    100.5;
NETWORK
TITLE =

      A(    ;
      O     I    113.3;
      O     I    317.3;
      )     ;
      AN    Q    100.0;
      AN    Q    100.1;
      =     Q    100.3;
NETWORK
TITLE =리턴2 인버터 인터록

NETWORK
TITLE =

      A     M   1046.0;
      =     L      0.0;
      A     L      0.0;
      BLD   102;
      =     Q    284.0;
      A     L      0.0;
      AN    M   1046.6;
      =     Q    284.4;
      A     L      0.0;
      A     M   1046.6;
      =     Q    284.5;
NETWORK
TITLE =

      A     I    113.3;
      AN    Q    284.0;
      =     Q    284.3;
NETWORK
TITLE =
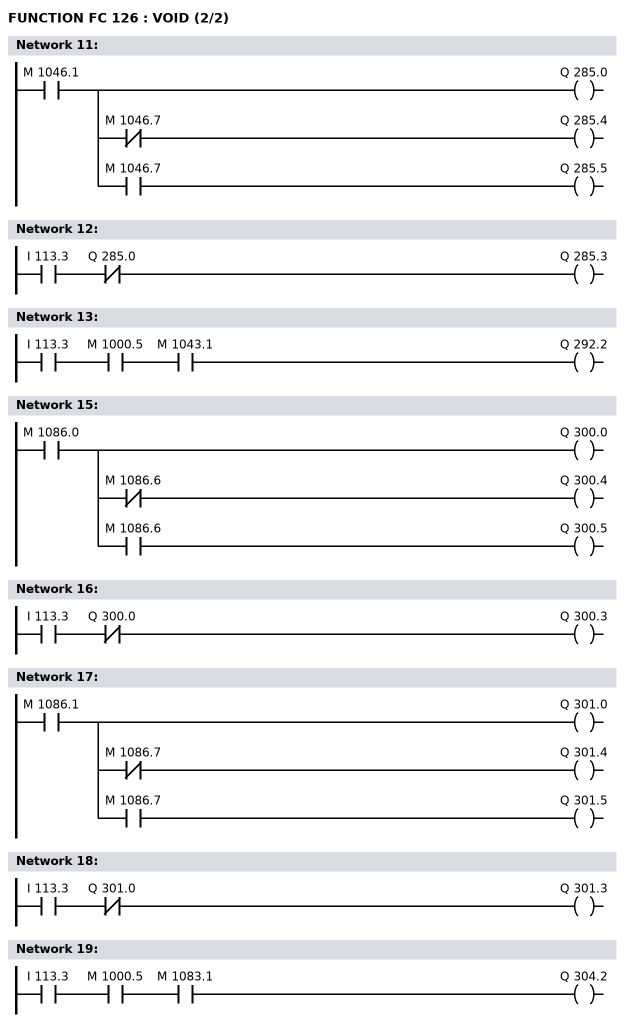

      A     M   1046.1;
      =     L      0.0;
      A     L      0.0;
      BLD   102;
      =     Q    285.0;
      A     L      0.0;
      AN    M   1046.7;
      =     Q    285.4;
      A     L      0.0;
      A     M   1046.7;
      =     Q    285.5;
NETWORK
TITLE =

      A     I    113.3;
      AN    Q    285.0;
      =     Q    285.3;
NETWORK
TITLE =

      A     I    113.3;
      A     M   1000.5;
      A     M   1043.1;
      =     Q    292.2;
NETWORK
TITLE =리턴3 인버터 인터록

NETWORK
TITLE =

      A     M   1086.0;
      =     L      0.0;
      A     L      0.0;
      BLD   102;
      =     Q    300.0;
      A     L      0.0;
      AN    M   1086.6;
      =     Q    300.4;
      A     L      0.0;
      A     M   1086.6;
      =     Q    300.5;
NETWORK
TITLE =

      A     I    113.3;
      AN    Q    300.0;
      =     Q    300.3;
NETWORK
TITLE =

      A     M   1086.1;
      =     L      0.0;
      A     L      0.0;
      BLD   102;
      =     Q    301.0;
      A     L      0.0;
      AN    M   1086.7;
      =     Q    301.4;
      A     L      0.0;
      A     M   1086.7;
      =     Q    301.5;
NETWORK
TITLE =

      A     I    113.3;
      AN    Q    301.0;
      =     Q    301.3;
NETWORK
TITLE =

      A     I    113.3;
      A     M   1000.5;
      A     M   1083.1;
      =     Q    304.2;
END_FUNCTION

FUNCTION_BLOCK FB 130
TITLE =
VERSION : 0.1


VAR
  S_IN_TRV_MODE : FB 402;
END_VAR
BEGIN
NETWORK
TITLE =
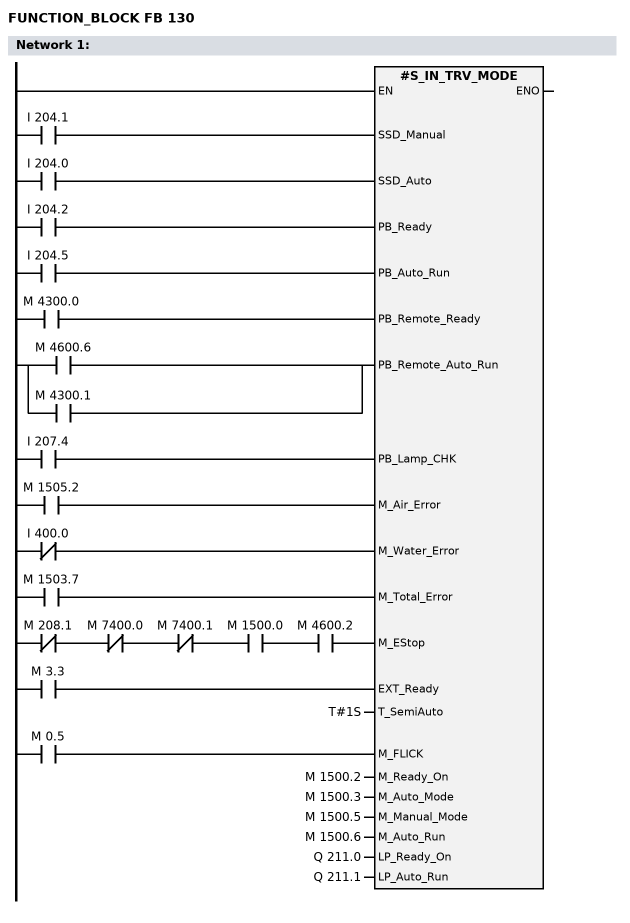

      A     I    204.1;
      =     L      0.0;
      BLD   103;
      A     I    204.0;
      =     L      0.1;
      BLD   103;
      A     I    204.2;
      =     L      0.2;
      BLD   103;
      A     I    204.5;
      =     L      0.3;
      BLD   103;
      A     M   4300.0;
      =     L      0.4;
      BLD   103;
      A(    ;
      O     M   4600.6;
      O     M   4300.1;
      )     ;
      =     L      0.5;
      BLD   103;
      A     I    207.4;
      =     L      0.6;
      BLD   103;
      A     M   1505.2;
      =     L      0.7;
      BLD   103;
      AN    I    400.0;
      =     L      1.0;
      BLD   103;
      A     M   1503.7;
      =     L      1.1;
      BLD   103;
      AN    M    208.1;
      AN    M   7400.0;
      AN    M   7400.1;
      A     M   1500.0;
      A     M   4600.2;
      =     L      1.2;
      BLD   103;
      A     M      3.3;
      =     L      1.3;
      BLD   103;
      A     M      0.5;
      =     L      1.5;
      BLD   103;
      CALL #S_IN_TRV_MODE (
           SSD_Manual               := L      0.0,
           SSD_Auto                 := L      0.1,
           PB_Ready                 := L      0.2,
           PB_Auto_Run              := L      0.3,
           PB_Remote_Ready          := L      0.4,
           PB_Remote_Auto_Run       := L      0.5,
           PB_Lamp_CHK              := L      0.6,
           M_Air_Error              := L      0.7,
           M_Water_Error            := L      1.0,
           M_Total_Error            := L      1.1,
           M_EStop                  := L      1.2,
           EXT_Ready                := L      1.3,
           T_SemiAuto               := T#1S,
           M_FLICK                  := L      1.5,
           M_Ready_On               := M   1500.2,
           M_Auto_Mode              := M   1500.3,
           M_Manual_Mode            := M   1500.5,
           M_Auto_Run               := M   1500.6,
           LP_Ready_On              := Q    211.0,
           LP_Auto_Run              := Q    211.1);
      NOP   0;
END_FUNCTION_BLOCK

DATA_BLOCK DB 130
TITLE =
VERSION : 0.0

 FB 130
BEGIN
   S_IN_TRV_MODE.SSD_Manual := FALSE;
   S_IN_TRV_MODE.SSD_Auto := FALSE;
   S_IN_TRV_MODE.PB_Ready := FALSE;
   S_IN_TRV_MODE.PB_Auto_Run := FALSE;
   S_IN_TRV_MODE.PB_Remote_Ready := FALSE;
   S_IN_TRV_MODE.PB_Remote_Auto_Run := FALSE;
   S_IN_TRV_MODE.PB_Lamp_CHK := FALSE;
   S_IN_TRV_MODE.M_Air_Error := FALSE;
   S_IN_TRV_MODE.M_Water_Error := FALSE;
   S_IN_TRV_MODE.M_Total_Error := FALSE;
   S_IN_TRV_MODE.M_EStop := FALSE;
   S_IN_TRV_MODE.EXT_Ready := FALSE;
   S_IN_TRV_MODE.EXT_Auto := FALSE;
   S_IN_TRV_MODE.T_SemiAuto := T#0MS;
   S_IN_TRV_MODE.M_FLICK := FALSE;
   S_IN_TRV_MODE.M_Ready_On := FALSE;
   S_IN_TRV_MODE.M_Auto_Mode := FALSE;
   S_IN_TRV_MODE.M_SemiAuto_Mode := FALSE;
   S_IN_TRV_MODE.M_Manual_Mode := FALSE;
   S_IN_TRV_MODE.M_Auto_Run := FALSE;
   S_IN_TRV_MODE.LP_Ready_On := FALSE;
   S_IN_TRV_MODE.LP_Auto_Run := FALSE;
   S_IN_TRV_MODE.AUTO_MODE_DELAY.IN := FALSE;
   S_IN_TRV_MODE.AUTO_MODE_DELAY.PT := T#0MS;
   S_IN_TRV_MODE.AUTO_MODE_DELAY.Q := FALSE;
   S_IN_TRV_MODE.AUTO_MODE_DELAY.ET := T#0MS;
   S_IN_TRV_MODE.AUTO_MODE_DELAY.STATE := B#16#0;
   S_IN_TRV_MODE.AUTO_MODE_DELAY.STIME := T#0MS;
   S_IN_TRV_MODE.AUTO_MODE_DELAY.ATIME := T#0MS;
   S_IN_TRV_MODE.SEMI_AUTO_DELAY.IN := FALSE;
   S_IN_TRV_MODE.SEMI_AUTO_DELAY.PT := T#0MS;
   S_IN_TRV_MODE.SEMI_AUTO_DELAY.Q := FALSE;
   S_IN_TRV_MODE.SEMI_AUTO_DELAY.ET := T#0MS;
   S_IN_TRV_MODE.SEMI_AUTO_DELAY.STATE := B#16#0;
   S_IN_TRV_MODE.SEMI_AUTO_DELAY.STIME := T#0MS;
   S_IN_TRV_MODE.SEMI_AUTO_DELAY.ATIME := T#0MS;
   S_IN_TRV_MODE.MANUAL_DELAY.IN := FALSE;
   S_IN_TRV_MODE.MANUAL_DELAY.PT := T#0MS;
   S_IN_TRV_MODE.MANUAL_DELAY.Q := FALSE;
   S_IN_TRV_MODE.MANUAL_DELAY.ET := T#0MS;
   S_IN_TRV_MODE.MANUAL_DELAY.STATE := B#16#0;
   S_IN_TRV_MODE.MANUAL_DELAY.STIME := T#0MS;
   S_IN_TRV_MODE.MANUAL_DELAY.ATIME := T#0MS;
END_DATA_BLOCK

FUNCTION FC 130 : VOID
TITLE =
VERSION : 0.1

BEGIN
NETWORK
TITLE =
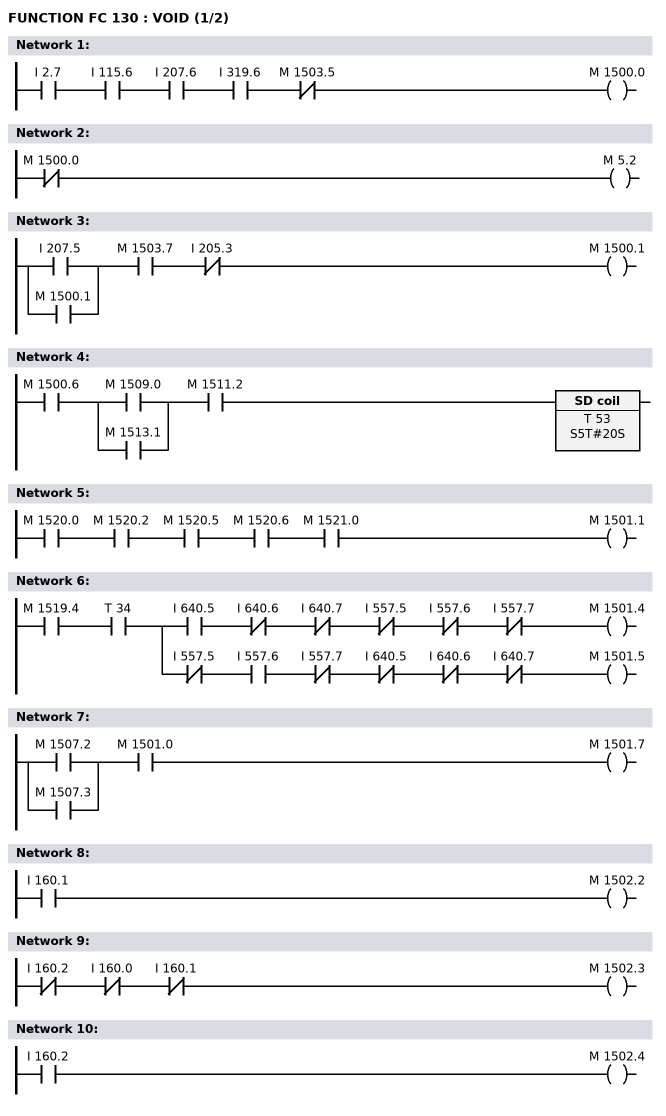

      A     I      2.7;
      A     I    115.6;
      A     I    207.6;
      A     I    319.6;
      AN    M   1503.5;
      =     M   1500.0;
NETWORK
TITLE =

      AN    M   1500.0;
      =     M      5.2;
NETWORK
TITLE =

      A(    ;
      O     I    207.5;
      O     M   1500.1;
      )     ;
      A     M   1503.7;
      AN    I    205.3;
      =     M   1500.1;
NETWORK
TITLE =

      A     M   1500.6;
      A(    ;
      O     M   1509.0;
      O     M   1513.1;
      )     ;
      A     M   1511.2;
      L     S5T#20S;
      SD    T     53;
NETWORK
TITLE =

      A     M   1520.0;
      A     M   1520.2;
      A     M   1520.5;
      A     M   1520.6;
      A     M   1521.0;
      =     M   1501.1;
NETWORK
TITLE =

      A     M   1519.4;
      A     T     34;
      =     L      0.0;
      A     L      0.0;
      A     I    640.5;
      AN    I    640.6;
      AN    I    640.7;
      AN    I    557.5;
      AN    I    557.6;
      AN    I    557.7;
      =     M   1501.4;
      A     L      0.0;
      AN    I    557.5;
      A     I    557.6;
      AN    I    557.7;
      AN    I    640.5;
      AN    I    640.6;
      AN    I    640.7;
      =     M   1501.5;
NETWORK
TITLE =

      A(    ;
      O     M   1507.2;
      O     M   1507.3;
      )     ;
      A     M   1501.0;
      =     M   1501.7;
NETWORK
TITLE =

      A     I    160.1;
      =     M   1502.2;
NETWORK
TITLE =

      AN    I    160.2;
      AN    I    160.0;
      AN    I    160.1;
      =     M   1502.3;
NETWORK
TITLE =

      A     I    160.2;
      =     M   1502.4;
NETWORK
TITLE =
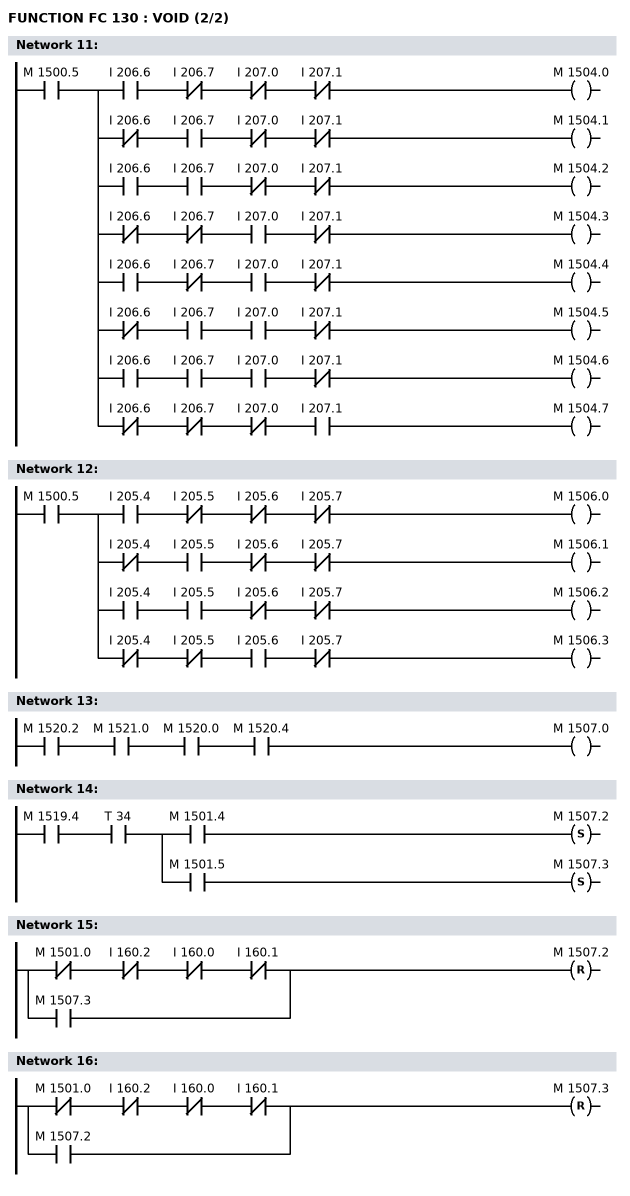

      A     M   1500.5;
      =     L      0.0;
      A     L      0.0;
      A     I    206.6;
      AN    I    206.7;
      AN    I    207.0;
      AN    I    207.1;
      =     M   1504.0;
      A     L      0.0;
      AN    I    206.6;
      A     I    206.7;
      AN    I    207.0;
      AN    I    207.1;
      =     M   1504.1;
      A     L      0.0;
      A     I    206.6;
      A     I    206.7;
      AN    I    207.0;
      AN    I    207.1;
      =     M   1504.2;
      A     L      0.0;
      AN    I    206.6;
      AN    I    206.7;
      A     I    207.0;
      AN    I    207.1;
      =     M   1504.3;
      A     L      0.0;
      A     I    206.6;
      AN    I    206.7;
      A     I    207.0;
      AN    I    207.1;
      =     M   1504.4;
      A     L      0.0;
      AN    I    206.6;
      A     I    206.7;
      A     I    207.0;
      AN    I    207.1;
      =     M   1504.5;
      A     L      0.0;
      A     I    206.6;
      A     I    206.7;
      A     I    207.0;
      AN    I    207.1;
      =     M   1504.6;
      A     L      0.0;
      AN    I    206.6;
      AN    I    206.7;
      AN    I    207.0;
      A     I    207.1;
      =     M   1504.7;
NETWORK
TITLE =

      A     M   1500.5;
      =     L      0.0;
      A     L      0.0;
      A     I    205.4;
      AN    I    205.5;
      AN    I    205.6;
      AN    I    205.7;
      =     M   1506.0;
      A     L      0.0;
      AN    I    205.4;
      A     I    205.5;
      AN    I    205.6;
      AN    I    205.7;
      =     M   1506.1;
      A     L      0.0;
      A     I    205.4;
      A     I    205.5;
      AN    I    205.6;
      AN    I    205.7;
      =     M   1506.2;
      A     L      0.0;
      AN    I    205.4;
      AN    I    205.5;
      A     I    205.6;
      AN    I    205.7;
      =     M   1506.3;
NETWORK
TITLE =

      A     M   1520.2;
      A     M   1521.0;
      A     M   1520.0;
      A     M   1520.4;
      =     M   1507.0;
NETWORK
TITLE =

      A     M   1519.4;
      A     T     34;
      =     L      0.0;
      A     L      0.0;
      A     M   1501.4;
      S     M   1507.2;
      A     L      0.0;
      A     M   1501.5;
      S     M   1507.3;
NETWORK
TITLE =

      AN    M   1501.0;
      AN    I    160.2;
      AN    I    160.0;
      AN    I    160.1;
      O     M   1507.3;
      R     M   1507.2;
NETWORK
TITLE =

      AN    M   1501.0;
      AN    I    160.2;
      AN    I    160.0;
      AN    I    160.1;
      O     M   1507.2;
      R     M   1507.3;
NETWORK
TITLE =

      AN    OV;
      =     L      0.0;
      A     L      0.0;
      A     M   1513.1;
      S     M   1507.6;
      A     L      0.0;
      A(    ;
      O     M   1513.3;
      O     M   1513.2;
      )     ;
      R     M   1507.6;
NETWORK
TITLE =

      A     M   1507.6;
      AN    M   1502.3;
      =     M   1507.7;
END_FUNCTION

FUNCTION_BLOCK FB 131
TITLE =
VERSION : 0.1


VAR
  IN_TRV_CUSHION_B : FB 424;
  IN_TRV_GUIDE : FB 424;
  IN_TRV_CLAMP : FB 424;
  IN_TRV_STOPPER : FB 424;
  IN_TRV_LIFT1 : FB 424;
  IN_TRV_ELE : FB 424;
  IN_TRV_LIFT2 : FB 424;
  IN_TRV_ELE_AIR : FB 424;
END_VAR
BEGIN
NETWORK
TITLE =
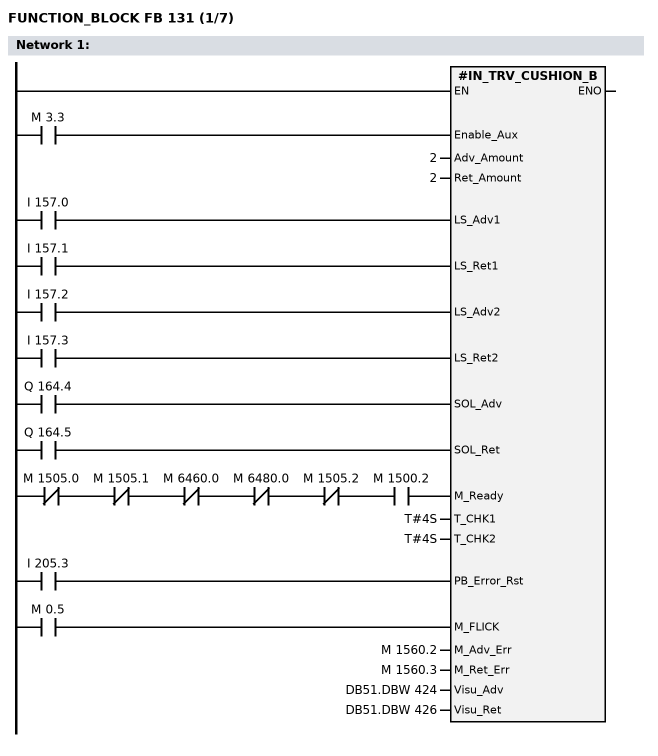

      A     M      3.3;
      =     L      0.0;
      BLD   103;
      A     I    157.0;
      =     L      0.1;
      BLD   103;
      A     I    157.1;
      =     L      0.2;
      BLD   103;
      A     I    157.2;
      =     L      0.3;
      BLD   103;
      A     I    157.3;
      =     L      0.4;
      BLD   103;
      A     Q    164.4;
      =     L      1.1;
      BLD   103;
      A     Q    164.5;
      =     L      1.2;
      BLD   103;
      AN    M   1505.0;
      AN    M   1505.1;
      AN    M   6460.0;
      AN    M   6480.0;
      AN    M   1505.2;
      A     M   1500.2;
      =     L      1.3;
      BLD   103;
      A     I    205.3;
      =     L      1.5;
      BLD   103;
      A     M      0.5;
      =     L      1.6;
      BLD   103;
      CALL #IN_TRV_CUSHION_B (
           Enable_Aux               := L      0.0,
           Adv_Amount               := 2,
           Ret_Amount               := 2,
           LS_Adv1                  := L      0.1,
           LS_Ret1                  := L      0.2,
           LS_Adv2                  := L      0.3,
           LS_Ret2                  := L      0.4,
           SOL_Adv                  := L      1.1,
           SOL_Ret                  := L      1.2,
           M_Ready                  := L      1.3,
           T_CHK1                   := T#4S,
           T_CHK2                   := T#4S,
           PB_Error_Rst             := L      1.5,
           M_FLICK                  := L      1.6,
           M_Adv_Err                := M   1560.2,
           M_Ret_Err                := M   1560.3,
           Visu_Adv                 := DB51.DBW  424,
           Visu_Ret                 := DB51.DBW  426);
      NOP   0;
NETWORK
TITLE =
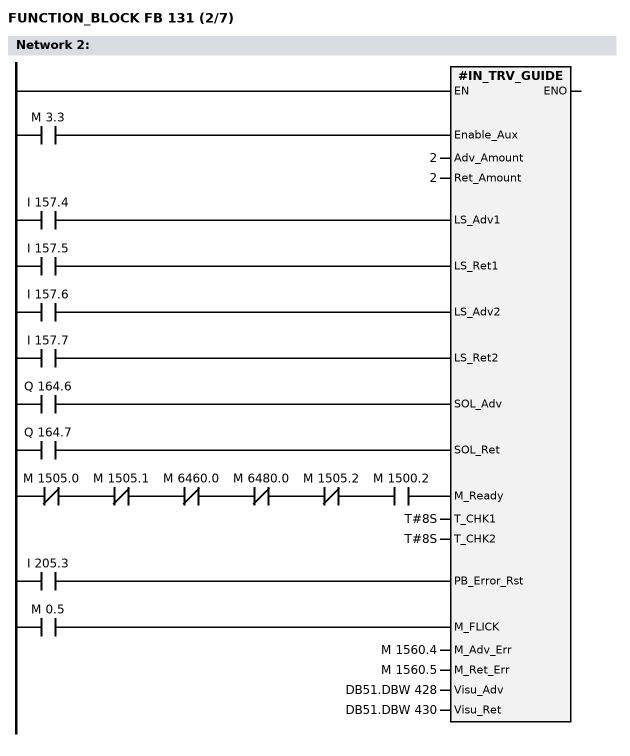

      A     M      3.3;
      =     L      0.0;
      BLD   103;
      A     I    157.4;
      =     L      0.1;
      BLD   103;
      A     I    157.5;
      =     L      0.2;
      BLD   103;
      A     I    157.6;
      =     L      0.3;
      BLD   103;
      A     I    157.7;
      =     L      0.4;
      BLD   103;
      A     Q    164.6;
      =     L      1.1;
      BLD   103;
      A     Q    164.7;
      =     L      1.2;
      BLD   103;
      AN    M   1505.0;
      AN    M   1505.1;
      AN    M   6460.0;
      AN    M   6480.0;
      AN    M   1505.2;
      A     M   1500.2;
      =     L      1.3;
      BLD   103;
      A     I    205.3;
      =     L      1.5;
      BLD   103;
      A     M      0.5;
      =     L      1.6;
      BLD   103;
      CALL #IN_TRV_GUIDE (
           Enable_Aux               := L      0.0,
           Adv_Amount               := 2,
           Ret_Amount               := 2,
           LS_Adv1                  := L      0.1,
           LS_Ret1                  := L      0.2,
           LS_Adv2                  := L      0.3,
           LS_Ret2                  := L      0.4,
           SOL_Adv                  := L      1.1,
           SOL_Ret                  := L      1.2,
           M_Ready                  := L      1.3,
           T_CHK1                   := T#8S,
           T_CHK2                   := T#8S,
           PB_Error_Rst             := L      1.5,
           M_FLICK                  := L      1.6,
           M_Adv_Err                := M   1560.4,
           M_Ret_Err                := M   1560.5,
           Visu_Adv                 := DB51.DBW  428,
           Visu_Ret                 := DB51.DBW  430);
      NOP   0;
NETWORK
TITLE =
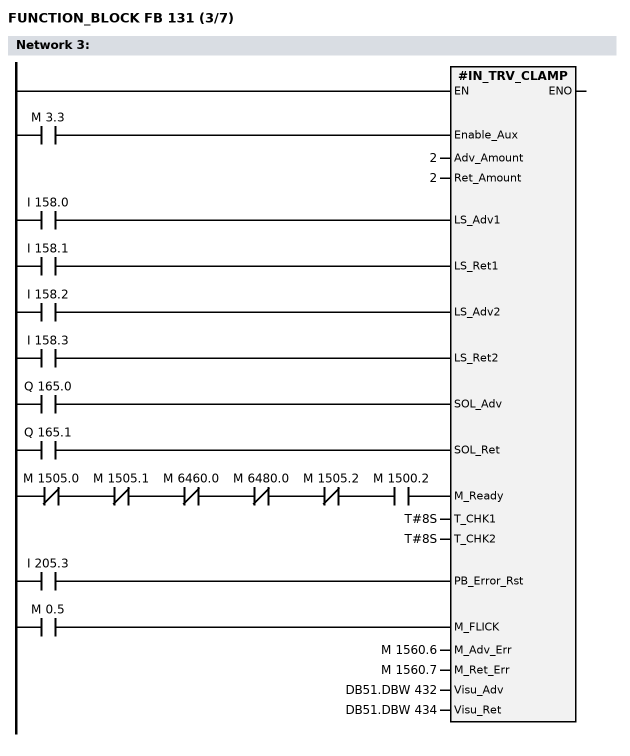

      A     M      3.3;
      =     L      0.0;
      BLD   103;
      A     I    158.0;
      =     L      0.1;
      BLD   103;
      A     I    158.1;
      =     L      0.2;
      BLD   103;
      A     I    158.2;
      =     L      0.3;
      BLD   103;
      A     I    158.3;
      =     L      0.4;
      BLD   103;
      A     Q    165.0;
      =     L      1.1;
      BLD   103;
      A     Q    165.1;
      =     L      1.2;
      BLD   103;
      AN    M   1505.0;
      AN    M   1505.1;
      AN    M   6460.0;
      AN    M   6480.0;
      AN    M   1505.2;
      A     M   1500.2;
      =     L      1.3;
      BLD   103;
      A     I    205.3;
      =     L      1.5;
      BLD   103;
      A     M      0.5;
      =     L      1.6;
      BLD   103;
      CALL #IN_TRV_CLAMP (
           Enable_Aux               := L      0.0,
           Adv_Amount               := 2,
           Ret_Amount               := 2,
           LS_Adv1                  := L      0.1,
           LS_Ret1                  := L      0.2,
           LS_Adv2                  := L      0.3,
           LS_Ret2                  := L      0.4,
           SOL_Adv                  := L      1.1,
           SOL_Ret                  := L      1.2,
           M_Ready                  := L      1.3,
           T_CHK1                   := T#8S,
           T_CHK2                   := T#8S,
           PB_Error_Rst             := L      1.5,
           M_FLICK                  := L      1.6,
           M_Adv_Err                := M   1560.6,
           M_Ret_Err                := M   1560.7,
           Visu_Adv                 := DB51.DBW  432,
           Visu_Ret                 := DB51.DBW  434);
      NOP   0;
NETWORK
TITLE =
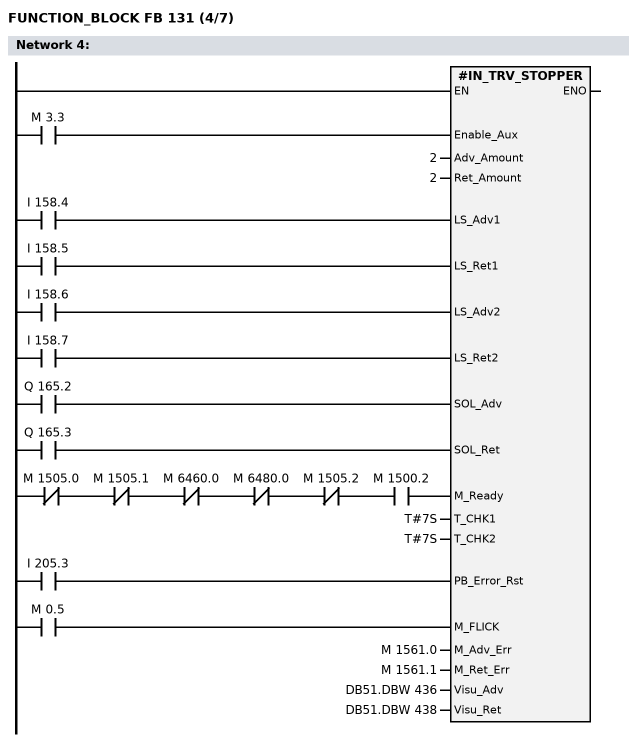

      A     M      3.3;
      =     L      0.0;
      BLD   103;
      A     I    158.4;
      =     L      0.1;
      BLD   103;
      A     I    158.5;
      =     L      0.2;
      BLD   103;
      A     I    158.6;
      =     L      0.3;
      BLD   103;
      A     I    158.7;
      =     L      0.4;
      BLD   103;
      A     Q    165.2;
      =     L      1.1;
      BLD   103;
      A     Q    165.3;
      =     L      1.2;
      BLD   103;
      AN    M   1505.0;
      AN    M   1505.1;
      AN    M   6460.0;
      AN    M   6480.0;
      AN    M   1505.2;
      A     M   1500.2;
      =     L      1.3;
      BLD   103;
      A     I    205.3;
      =     L      1.5;
      BLD   103;
      A     M      0.5;
      =     L      1.6;
      BLD   103;
      CALL #IN_TRV_STOPPER (
           Enable_Aux               := L      0.0,
           Adv_Amount               := 2,
           Ret_Amount               := 2,
           LS_Adv1                  := L      0.1,
           LS_Ret1                  := L      0.2,
           LS_Adv2                  := L      0.3,
           LS_Ret2                  := L      0.4,
           SOL_Adv                  := L      1.1,
           SOL_Ret                  := L      1.2,
           M_Ready                  := L      1.3,
           T_CHK1                   := T#7S,
           T_CHK2                   := T#7S,
           PB_Error_Rst             := L      1.5,
           M_FLICK                  := L      1.6,
           M_Adv_Err                := M   1561.0,
           M_Ret_Err                := M   1561.1,
           Visu_Adv                 := DB51.DBW  436,
           Visu_Ret                 := DB51.DBW  438);
      NOP   0;
NETWORK
TITLE =
